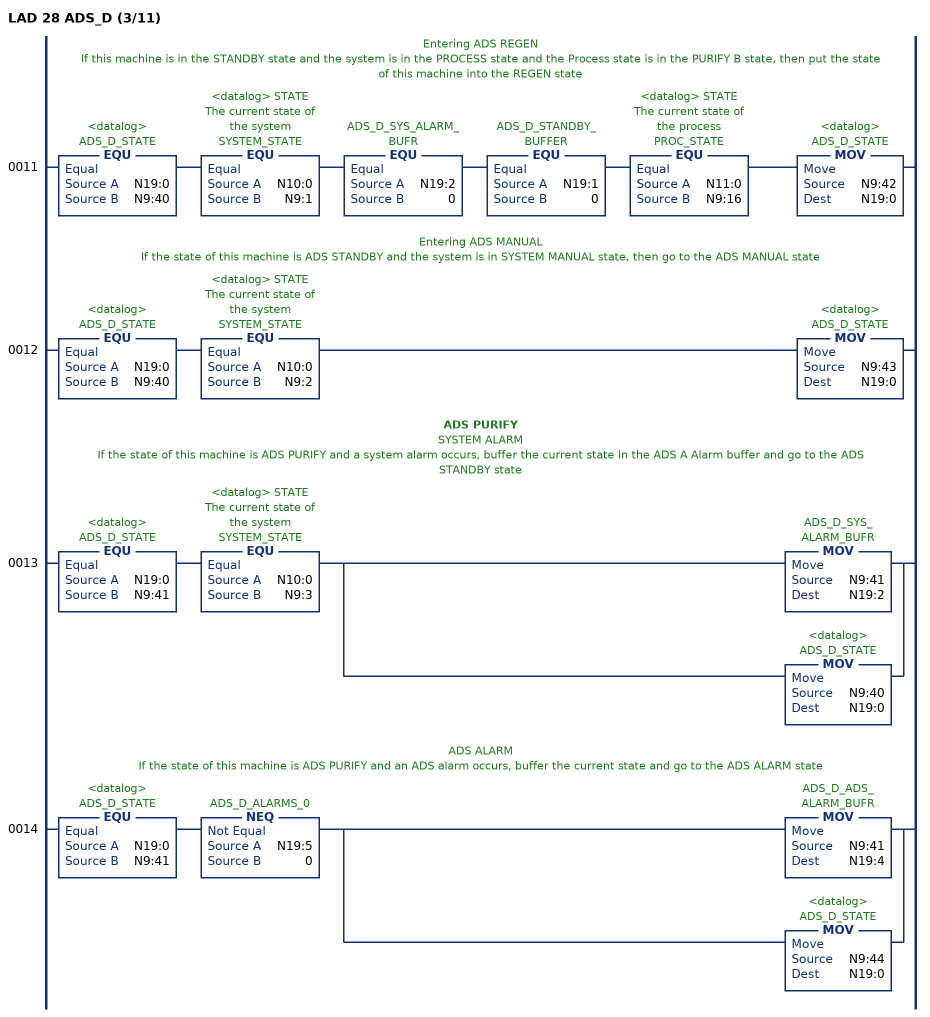
% Rung: 11 %
% Entering ADS REGEN
% If this machine is in the STANDBY state and the system is in the PROCESS state and the Process state is in the PURIFY B state, then put the state of this machine into the REGEN state %
SOR EQU N19:0 N9:40 EQU N10:0 N9:1 EQU N19:2 0 EQU N19:1 0 EQU N11:0 N9:16 MOV N9:42 N19:0 EOR
%   N19:0  ADS_D_STATE  "<datalog>" %
%   N9:40  ADS_STANDBY  "STATE ADS Standby" %
%   N10:0  SYSTEM_STATE  "<datalog> STATE The current state of the system" %
%   N9:1  SYSTEM_PROCESS  "STATE System Process" %
%   N19:2  ADS_D_SYS_ALARM_BUFR %
%   N19:1  ADS_D_STANDBY_BUFFER %
%   N11:0  PROC_STATE  "<datalog> STATE The current state of the process" %
%   N9:16  PROC_REGEN_D  "STATE Process Regen D" %
%   N9:42  ADS_REGEN  "STATE ADS Regen" %
% Rung: 12 %
% Entering ADS MANUAL
% If the state of this machine is ADS STANDBY and the system is in SYSTEM MANUAL state, then go to the ADS MANUAL state %
SOR EQU N19:0 N9:40 EQU N10:0 N9:2 MOV N9:43 N19:0 EOR
%   N19:0  ADS_D_STATE  "<datalog>" %
%   N9:40  ADS_STANDBY  "STATE ADS Standby" %
%   N10:0  SYSTEM_STATE  "<datalog> STATE The current state of the system" %
%   N9:2  SYSTEM_MANUAL  "STATE System Manual" %
%   N9:43  ADS_MANUAL  "STATE ADS Manual" %
% Rung: 13 %
% TITLE: ADS PURIFY %
% SYSTEM ALARM
% If the state of this machine is ADS PURIFY and a system alarm occurs, buffer the current state in the ADS A Alarm buffer and go to the ADS STANDBY state %
SOR EQU N19:0 N9:41 EQU N10:0 N9:3 BST MOV N9:41 N19:2 NXB MOV N9:40 N19:0 BND EOR
%   N19:0  ADS_D_STATE  "<datalog>" %
%   N9:41  ADS_PURIFY  "STATE ADS Purify" %
%   N10:0  SYSTEM_STATE  "<datalog> STATE The current state of the system" %
%   N9:3  SYSTEM_ALARM  "STATE System Alarm" %
%   N19:2  ADS_D_SYS_ALARM_BUFR %
%   N9:40  ADS_STANDBY  "STATE ADS Standby" %
% Rung: 14 %
% ADS ALARM
% If the state of this machine is ADS PURIFY and an ADS alarm occurs, buffer the current state and go to the ADS ALARM state %
SOR EQU N19:0 N9:41 NEQ N19:5 0 BST MOV N9:41 N19:4 NXB MOV N9:44 N19:0 BND EOR
%   N19:0  ADS_D_STATE  "<datalog>" %
%   N9:41  ADS_PURIFY  "STATE ADS Purify" %
%   N19:5  ADS_D_ALARMS_0 %
%   N19:4  ADS_D_ADS_ALARM_BUFR %
%   N9:44  ADS_ALARM  "STATE ADS Alarm" %

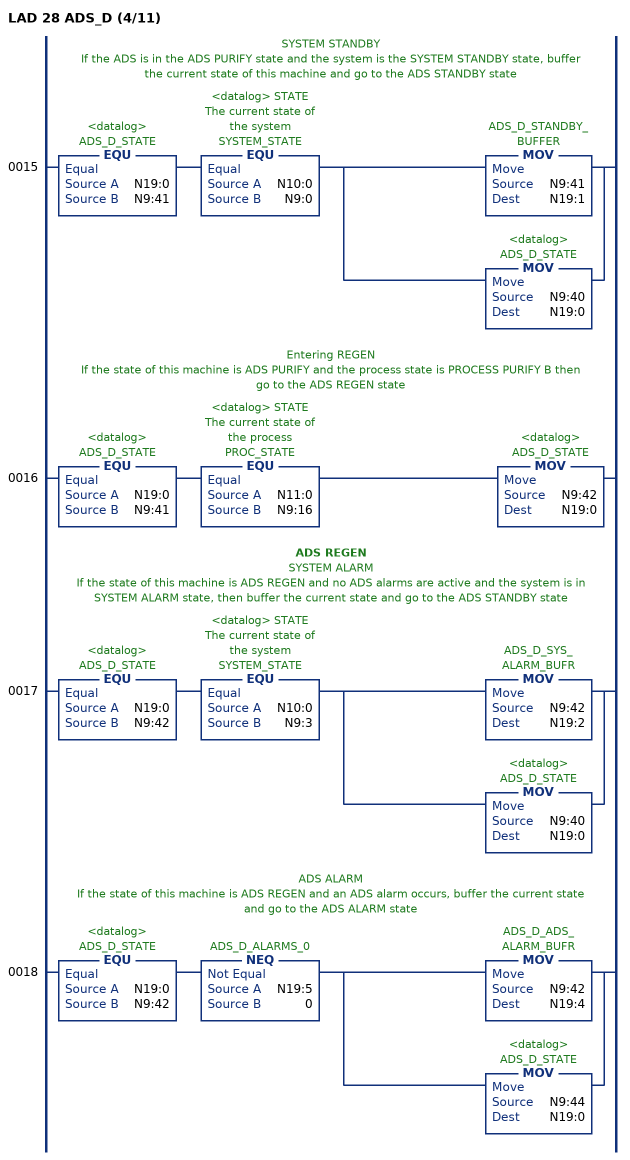
% Rung: 15 %
% SYSTEM STANDBY
% If the ADS is in the ADS PURIFY state and the system is the SYSTEM STANDBY state, buffer the current state of this machine and go to the ADS STANDBY state %
SOR EQU N19:0 N9:41 EQU N10:0 N9:0 BST MOV N9:41 N19:1 NXB MOV N9:40 N19:0 BND EOR
%   N19:0  ADS_D_STATE  "<datalog>" %
%   N9:41  ADS_PURIFY  "STATE ADS Purify" %
%   N10:0  SYSTEM_STATE  "<datalog> STATE The current state of the system" %
%   N9:0  SYSTEM_STANDBY  "STATE System Standby" %
%   N19:1  ADS_D_STANDBY_BUFFER %
%   N9:40  ADS_STANDBY  "STATE ADS Standby" %
% Rung: 16 %
% Entering REGEN
% If the state of this machine is ADS PURIFY and the process state is PROCESS PURIFY B then go to the ADS REGEN state %
SOR EQU N19:0 N9:41 EQU N11:0 N9:16 MOV N9:42 N19:0 EOR
%   N19:0  ADS_D_STATE  "<datalog>" %
%   N9:41  ADS_PURIFY  "STATE ADS Purify" %
%   N11:0  PROC_STATE  "<datalog> STATE The current state of the process" %
%   N9:16  PROC_REGEN_D  "STATE Process Regen D" %
%   N9:42  ADS_REGEN  "STATE ADS Regen" %
% Rung: 17 %
% TITLE: ADS REGEN %
% SYSTEM ALARM
% If the state of this machine is ADS REGEN and no ADS alarms are active and the system is in SYSTEM ALARM state, then buffer the current state and go to the ADS STANDBY state %
SOR EQU N19:0 N9:42 EQU N10:0 N9:3 BST MOV N9:42 N19:2 NXB MOV N9:40 N19:0 BND EOR
%   N19:0  ADS_D_STATE  "<datalog>" %
%   N9:42  ADS_REGEN  "STATE ADS Regen" %
%   N10:0  SYSTEM_STATE  "<datalog> STATE The current state of the system" %
%   N9:3  SYSTEM_ALARM  "STATE System Alarm" %
%   N19:2  ADS_D_SYS_ALARM_BUFR %
%   N9:40  ADS_STANDBY  "STATE ADS Standby" %
% Rung: 18 %
% ADS ALARM
% If the state of this machine is ADS REGEN and an ADS alarm occurs, buffer the current state and go to the ADS ALARM state %
SOR EQU N19:0 N9:42 NEQ N19:5 0 BST MOV N9:42 N19:4 NXB MOV N9:44 N19:0 BND EOR
%   N19:0  ADS_D_STATE  "<datalog>" %
%   N9:42  ADS_REGEN  "STATE ADS Regen" %
%   N19:5  ADS_D_ALARMS_0 %
%   N19:4  ADS_D_ADS_ALARM_BUFR %
%   N9:44  ADS_ALARM  "STATE ADS Alarm" %

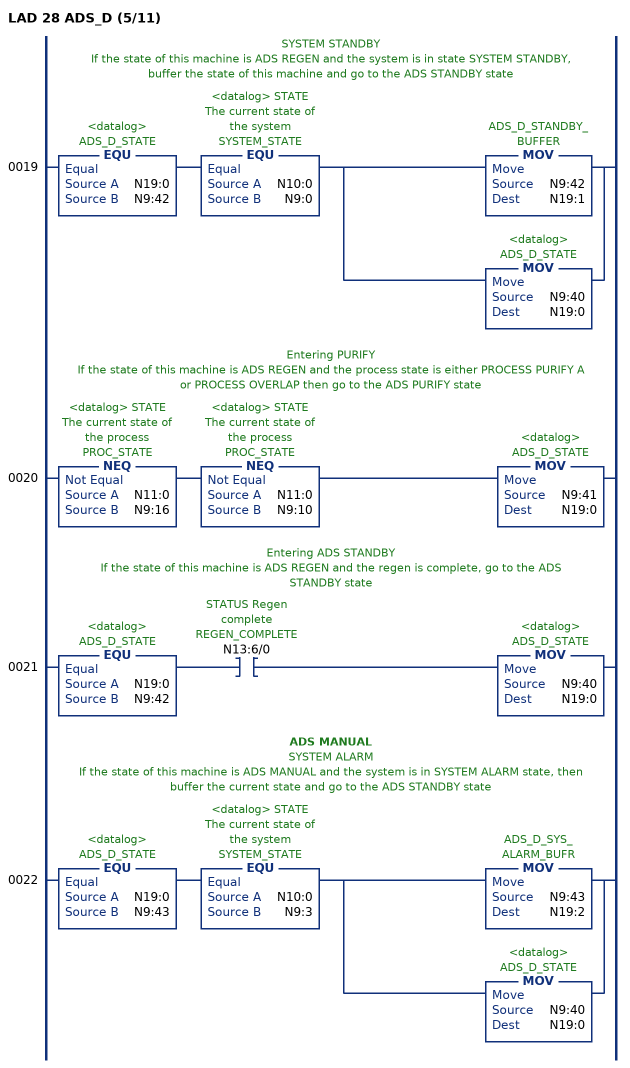
% Rung: 19 %
% SYSTEM STANDBY
% If the state of this machine is ADS REGEN and the system is in state SYSTEM STANDBY, buffer the state of this machine and go to the ADS STANDBY state %
SOR EQU N19:0 N9:42 EQU N10:0 N9:0 BST MOV N9:42 N19:1 NXB MOV N9:40 N19:0 BND EOR
%   N19:0  ADS_D_STATE  "<datalog>" %
%   N9:42  ADS_REGEN  "STATE ADS Regen" %
%   N10:0  SYSTEM_STATE  "<datalog> STATE The current state of the system" %
%   N9:0  SYSTEM_STANDBY  "STATE System Standby" %
%   N19:1  ADS_D_STANDBY_BUFFER %
%   N9:40  ADS_STANDBY  "STATE ADS Standby" %
% Rung: 20 %
% Entering PURIFY
% If the state of this machine is ADS REGEN and the process state is either PROCESS PURIFY A or PROCESS OVERLAP then go to the ADS PURIFY state %
SOR NEQ N11:0 N9:16 NEQ N11:0 N9:10 MOV N9:41 N19:0 EOR
%   N11:0  PROC_STATE  "<datalog> STATE The current state of the process" %
%   N9:16  PROC_REGEN_D  "STATE Process Regen D" %
%   N9:10  PROCESS_STANDBY  "STATE Process Standby" %
%   N9:41  ADS_PURIFY  "STATE ADS Purify" %
%   N19:0  ADS_D_STATE  "<datalog>" %
% Rung: 21 %
% Entering ADS STANDBY
% If the state of this machine is ADS REGEN and the regen is complete, go to the ADS STANDBY state %
SOR EQU N19:0 N9:42 XIC N13:6/0 MOV N9:40 N19:0 EOR
%   N19:0  ADS_D_STATE  "<datalog>" %
%   N9:42  ADS_REGEN  "STATE ADS Regen" %
%   N13:6/0  REGEN_COMPLETE  "STATUS Regen complete" %
%   N9:40  ADS_STANDBY  "STATE ADS Standby" %
% Rung: 22 %
% TITLE: ADS MANUAL %
% SYSTEM ALARM
% If the state of this machine is ADS MANUAL and the system is in SYSTEM ALARM state, then buffer the current state and go to the ADS STANDBY state %
SOR EQU N19:0 N9:43 EQU N10:0 N9:3 BST MOV N9:43 N19:2 NXB MOV N9:40 N19:0 BND EOR
%   N19:0  ADS_D_STATE  "<datalog>" %
%   N9:43  ADS_MANUAL  "STATE ADS Manual" %
%   N10:0  SYSTEM_STATE  "<datalog> STATE The current state of the system" %
%   N9:3  SYSTEM_ALARM  "STATE System Alarm" %
%   N19:2  ADS_D_SYS_ALARM_BUFR %
%   N9:40  ADS_STANDBY  "STATE ADS Standby" %

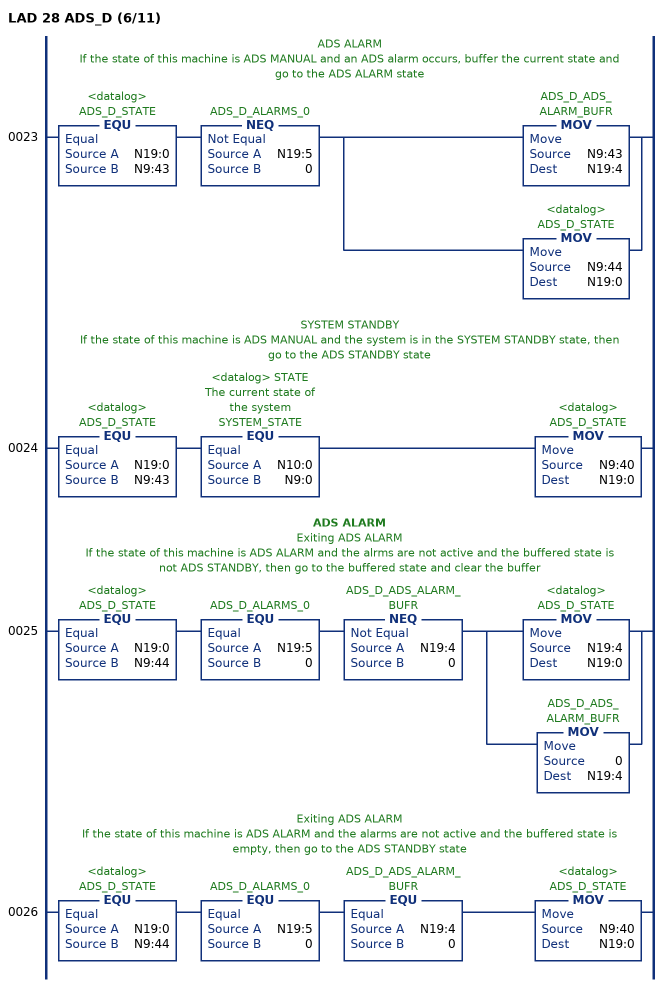
% Rung: 23 %
% ADS ALARM
% If the state of this machine is ADS MANUAL and an ADS alarm occurs, buffer the current state and go to the ADS ALARM state %
SOR EQU N19:0 N9:43 NEQ N19:5 0 BST MOV N9:43 N19:4 NXB MOV N9:44 N19:0 BND EOR
%   N19:0  ADS_D_STATE  "<datalog>" %
%   N9:43  ADS_MANUAL  "STATE ADS Manual" %
%   N19:5  ADS_D_ALARMS_0 %
%   N19:4  ADS_D_ADS_ALARM_BUFR %
%   N9:44  ADS_ALARM  "STATE ADS Alarm" %
% Rung: 24 %
% SYSTEM STANDBY
% If the state of this machine is ADS MANUAL and the system is in the SYSTEM STANDBY state, then go to the ADS STANDBY state %
SOR EQU N19:0 N9:43 EQU N10:0 N9:0 MOV N9:40 N19:0 EOR
%   N19:0  ADS_D_STATE  "<datalog>" %
%   N9:43  ADS_MANUAL  "STATE ADS Manual" %
%   N10:0  SYSTEM_STATE  "<datalog> STATE The current state of the system" %
%   N9:0  SYSTEM_STANDBY  "STATE System Standby" %
%   N9:40  ADS_STANDBY  "STATE ADS Standby" %
% Rung: 25 %
% TITLE: ADS ALARM %
% Exiting ADS ALARM
% If the state of this machine is ADS ALARM and the alrms are not active and the buffered state is not ADS STANDBY, then go to the buffered state and clear the buffer %
SOR EQU N19:0 N9:44 EQU N19:5 0 NEQ N19:4 0 BST MOV N19:4 N19:0 NXB MOV 0 N19:4 BND EOR
%   N19:0  ADS_D_STATE  "<datalog>" %
%   N9:44  ADS_ALARM  "STATE ADS Alarm" %
%   N19:5  ADS_D_ALARMS_0 %
%   N19:4  ADS_D_ADS_ALARM_BUFR %
% Rung: 26 %
% Exiting ADS ALARM
% If the state of this machine is ADS ALARM and the alarms are not active and the buffered state is empty, then go to the ADS STANDBY state %
SOR EQU N19:0 N9:44 EQU N19:5 0 EQU N19:4 0 MOV N9:40 N19:0 EOR
%   N19:0  ADS_D_STATE  "<datalog>" %
%   N9:44  ADS_ALARM  "STATE ADS Alarm" %
%   N19:5  ADS_D_ALARMS_0 %
%   N19:4  ADS_D_ADS_ALARM_BUFR %
%   N9:40  ADS_STANDBY  "STATE ADS Standby" %

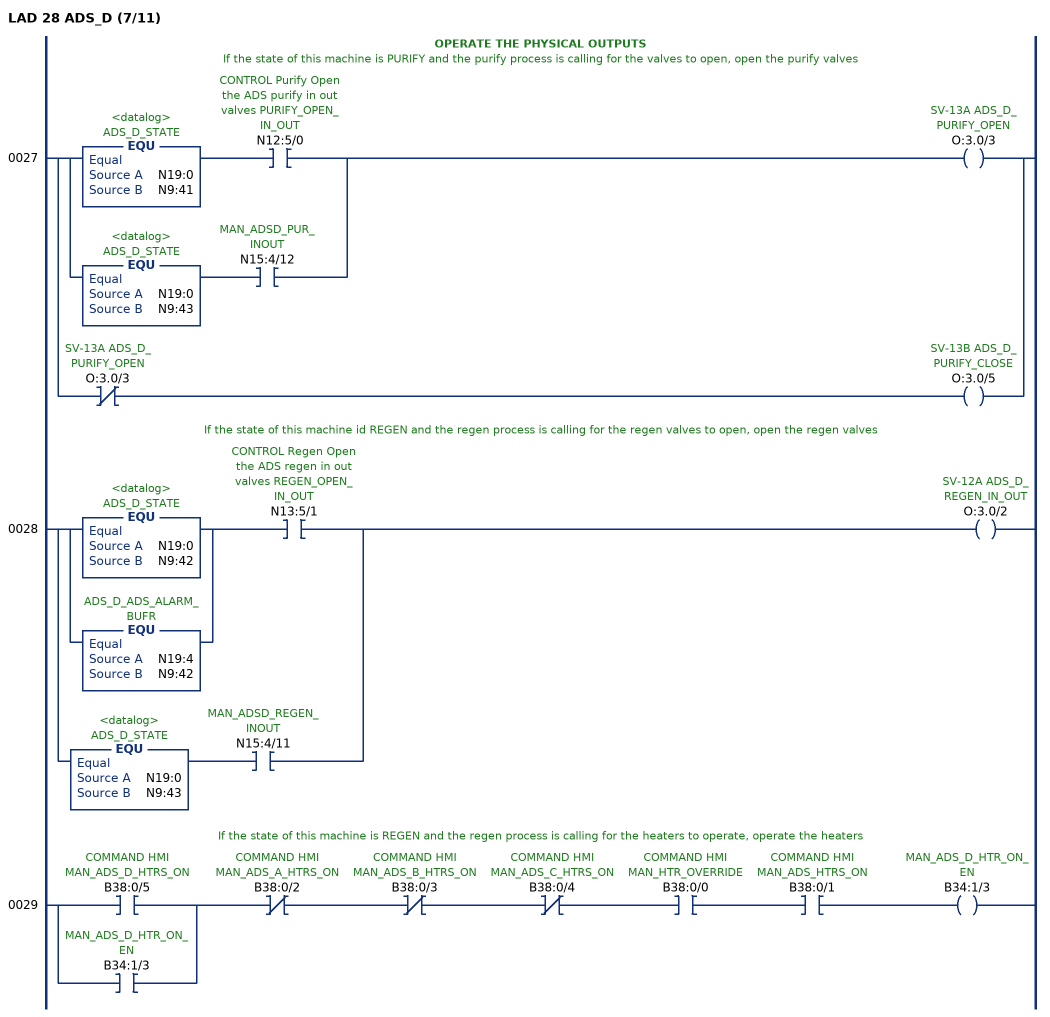
% Rung: 27 %
% TITLE: OPERATE THE PHYSICAL OUTPUTS %
% If the state of this machine is PURIFY and the purify process is calling for the valves to open, open the purify valves %
SOR BST BST EQU N19:0 N9:41 XIC N12:5/0 NXB EQU N19:0 N9:43 XIC N15:4/12 BND OTE O:3.0/3 NXB XIO O:3.0/3 OTE O:3.0/5 BND EOR
%   N19:0  ADS_D_STATE  "<datalog>" %
%   N9:41  ADS_PURIFY  "STATE ADS Purify" %
%   N12:5/0  PURIFY_OPEN_IN_OUT  "CONTROL Purify Open the ADS purify in out valves" %
%   N9:43  ADS_MANUAL  "STATE ADS Manual" %
%   N15:4/12  MAN_ADSD_PUR_INOUT %
%   O:3.0/3  ADS_D_PURIFY_OPEN  "SV-13A" %
%   O:3.0/5  ADS_D_PURIFY_CLOSE  "SV-13B" %
% Rung: 28 %
% If the state of this machine id REGEN and the regen process is calling for the regen valves to open, open the regen valves %
SOR BST BST EQU N19:0 N9:42 NXB EQU N19:4 N9:42 BND XIC N13:5/1 NXB EQU N19:0 N9:43 XIC N15:4/11 BND OTE O:3.0/2 EOR
%   N19:0  ADS_D_STATE  "<datalog>" %
%   N9:42  ADS_REGEN  "STATE ADS Regen" %
%   N19:4  ADS_D_ADS_ALARM_BUFR %
%   N13:5/1  REGEN_OPEN_IN_OUT  "CONTROL Regen Open the ADS regen in out valves" %
%   N9:43  ADS_MANUAL  "STATE ADS Manual" %
%   N15:4/11  MAN_ADSD_REGEN_INOUT %
%   O:3.0/2  ADS_D_REGEN_IN_OUT  "SV-12A" %
% Rung: 29 %
% If the state of this machine is REGEN and the regen process is calling for the heaters to operate, operate the heaters %
SOR BST XIC B38:0/5 NXB XIC B34:1/3 BND XIO B38:0/2 XIO B38:0/3 XIO B38:0/4 XIC B38:0/0 XIC B38:0/1 OTE B34:1/3 EOR
%   B38:0/5  MAN_ADS_D_HTRS_ON  "COMMAND HMI" %
%   B34:1/3  MAN_ADS_D_HTR_ON_EN %
%   B38:0/2  MAN_ADS_A_HTRS_ON  "COMMAND HMI" %
%   B38:0/3  MAN_ADS_B_HTRS_ON  "COMMAND HMI" %
%   B38:0/4  MAN_ADS_C_HTRS_ON  "COMMAND HMI" %
%   B38:0/0  MAN_HTR_OVERRIDE  "COMMAND HMI" %
%   B38:0/1  MAN_ADS_HTRS_ON  "COMMAND HMI" %

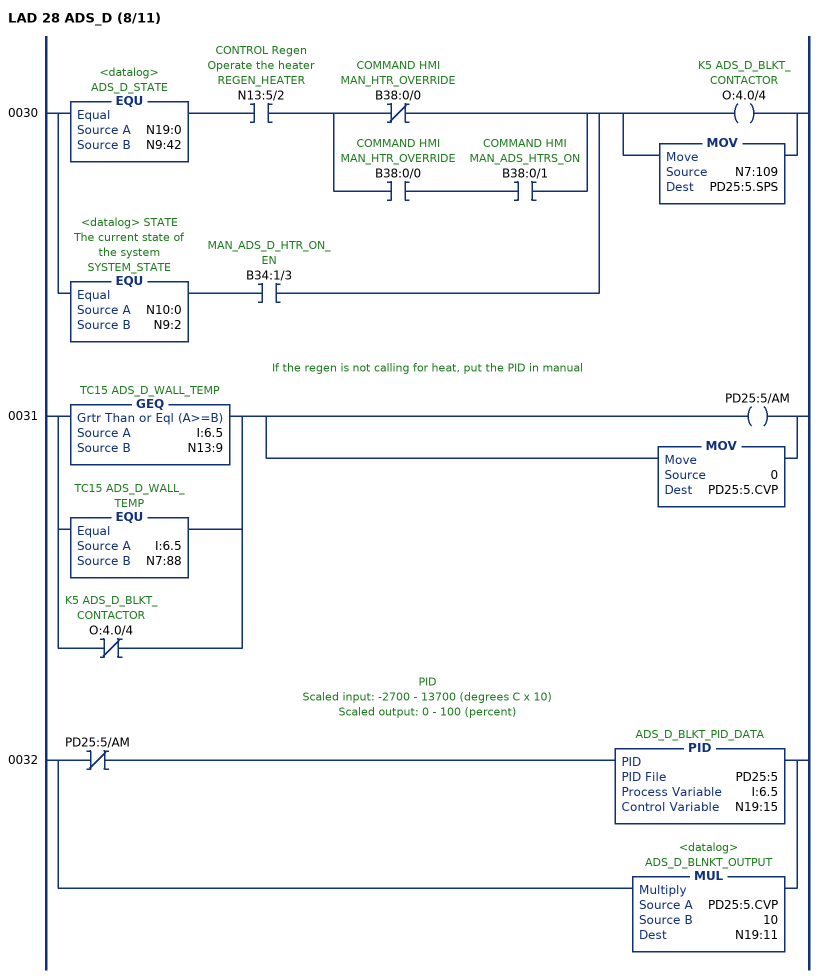
% Rung: 30 %
SOR BST EQU N19:0 N9:42 XIC N13:5/2 BST XIO B38:0/0 NXB XIC B38:0/0 XIC B38:0/1 BND NXB EQU N10:0 N9:2 XIC B34:1/3 BND BST OTE O:4.0/4 NXB MOV N7:109 PD25:5.SPS BND EOR
%   N19:0  ADS_D_STATE  "<datalog>" %
%   N9:42  ADS_REGEN  "STATE ADS Regen" %
%   N13:5/2  REGEN_HEATER  "CONTROL Regen Operate the heater" %
%   B38:0/0  MAN_HTR_OVERRIDE  "COMMAND HMI" %
%   B38:0/1  MAN_ADS_HTRS_ON  "COMMAND HMI" %
%   N10:0  SYSTEM_STATE  "<datalog> STATE The current state of the system" %
%   N9:2  SYSTEM_MANUAL  "STATE System Manual" %
%   B34:1/3  MAN_ADS_D_HTR_ON_EN %
%   O:4.0/4  ADS_D_BLKT_CONTACTOR  "K5" %
%   N7:109  BLANKET_SP  "<datalog> ADS Blanket PID Setpoint" %
% Rung: 31 %
% If the regen is not calling for heat, put the PID in manual %
SOR BST GEQ I:6.5 N13:9 NXB EQU I:6.5 N7:88 NXB XIO O:4.0/4 BND BST OTE PD25:5/AM NXB MOV 0 PD25:5.CVP BND EOR
%   I:6.5  ADS_D_WALL_TEMP  "TC15" %
%   N13:9  BLANKET_LIMIT  "ADS Blanket Temp Limit" %
%   N7:88  TC_OPEN_SP  "CONFIG TC Open Setpoint" %
%   O:4.0/4  ADS_D_BLKT_CONTACTOR  "K5" %
% Rung: 32 %
% PID
% Scaled input: -2700 - 13700 (degrees C x 10)
% Scaled output: 0 - 100 (percent) %
SOR BST XIO PD25:5/AM PID PD25:5 I:6.5 N19:15 NXB MUL PD25:5.CVP 10 N19:11 BND EOR
%   PD25:5  ADS_D_BLKT_PID_DATA %
%   I:6.5  ADS_D_WALL_TEMP  "TC15" %
%   N19:15  ADS_D_BLKT_OUTPT_RAW %
%   N19:11  ADS_D_BLNKT_OUTPUT  "<datalog>" %

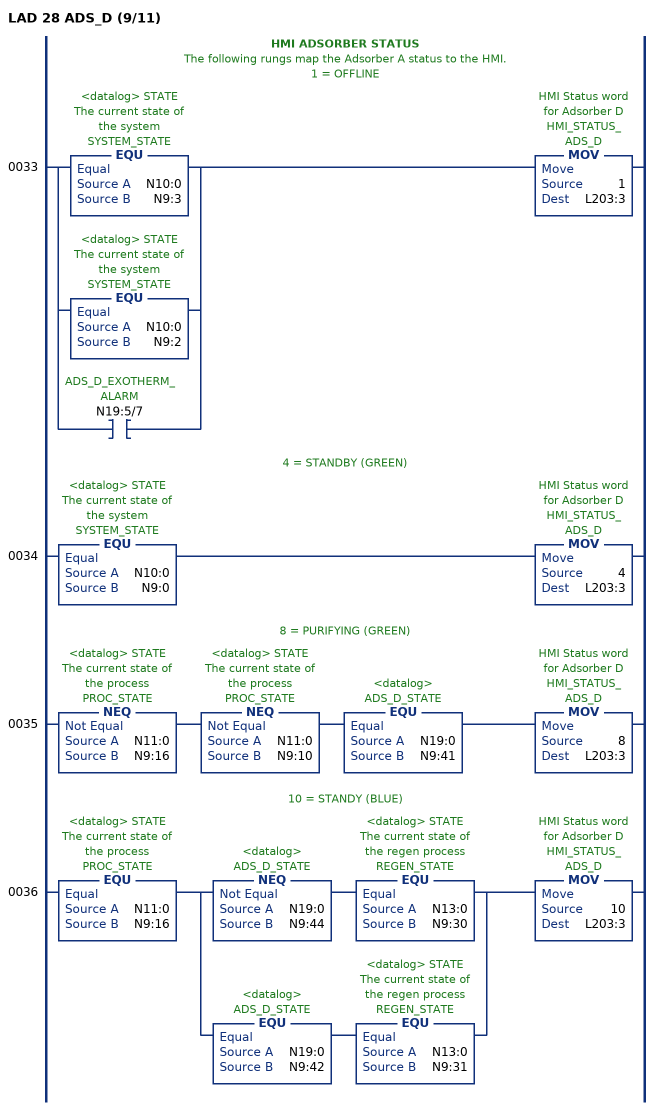
% Rung: 33 %
% TITLE: HMI ADSORBER STATUS %
% The following rungs map the Adsorber A status to the HMI.
% 1 = OFFLINE %
SOR BST EQU N10:0 N9:3 NXB EQU N10:0 N9:2 NXB XIC N19:5/7 BND MOV 1 L203:3 EOR
%   N10:0  SYSTEM_STATE  "<datalog> STATE The current state of the system" %
%   N9:3  SYSTEM_ALARM  "STATE System Alarm" %
%   N9:2  SYSTEM_MANUAL  "STATE System Manual" %
%   N19:5/7  ADS_D_EXOTHERM_ALARM %
%   L203:3  HMI_STATUS_ADS_D  "HMI Status word for Adsorber D" %
% Rung: 34 %
% 4 = STANDBY (GREEN) %
SOR EQU N10:0 N9:0 MOV 4 L203:3 EOR
%   N10:0  SYSTEM_STATE  "<datalog> STATE The current state of the system" %
%   N9:0  SYSTEM_STANDBY  "STATE System Standby" %
%   L203:3  HMI_STATUS_ADS_D  "HMI Status word for Adsorber D" %
% Rung: 35 %
% 8 = PURIFYING (GREEN) %
SOR NEQ N11:0 N9:16 NEQ N11:0 N9:10 EQU N19:0 N9:41 MOV 8 L203:3 EOR
%   N11:0  PROC_STATE  "<datalog> STATE The current state of the process" %
%   N9:16  PROC_REGEN_D  "STATE Process Regen D" %
%   N9:10  PROCESS_STANDBY  "STATE Process Standby" %
%   N19:0  ADS_D_STATE  "<datalog>" %
%   N9:41  ADS_PURIFY  "STATE ADS Purify" %
%   L203:3  HMI_STATUS_ADS_D  "HMI Status word for Adsorber D" %
% Rung: 36 %
% 10 = STANDY (BLUE) %
SOR EQU N11:0 N9:16 BST NEQ N19:0 N9:44 EQU N13:0 N9:30 NXB EQU N19:0 N9:42 EQU N13:0 N9:31 BND MOV 10 L203:3 EOR
%   N11:0  PROC_STATE  "<datalog> STATE The current state of the process" %
%   N9:16  PROC_REGEN_D  "STATE Process Regen D" %
%   N19:0  ADS_D_STATE  "<datalog>" %
%   N9:44  ADS_ALARM  "STATE ADS Alarm" %
%   N13:0  REGEN_STATE  "<datalog> STATE The current state of the regen process" %
%   N9:30  REGEN_STANDBY  "STATE Regen Standby" %
%   N9:42  ADS_REGEN  "STATE ADS Regen" %
%   N9:31  REGEN_DELAY  "STATE Regen Delay" %
%   L203:3  HMI_STATUS_ADS_D  "HMI Status word for Adsorber D" %

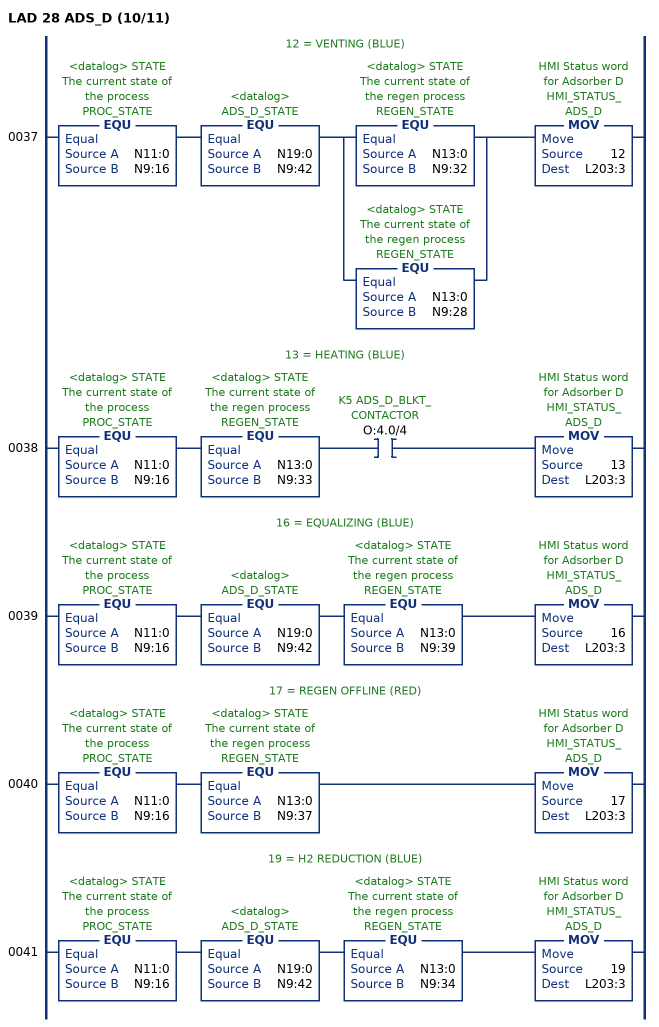
% Rung: 37 %
% 12 = VENTING (BLUE) %
SOR EQU N11:0 N9:16 EQU N19:0 N9:42 BST EQU N13:0 N9:32 NXB EQU N13:0 N9:28 BND MOV 12 L203:3 EOR
%   N11:0  PROC_STATE  "<datalog> STATE The current state of the process" %
%   N9:16  PROC_REGEN_D  "STATE Process Regen D" %
%   N19:0  ADS_D_STATE  "<datalog>" %
%   N9:42  ADS_REGEN  "STATE ADS Regen" %
%   N13:0  REGEN_STATE  "<datalog> STATE The current state of the regen process" %
%   N9:32  REGEN_VENT  "STATE Regen Vent" %
%   N9:28  REGEN_VENT_2 %
%   L203:3  HMI_STATUS_ADS_D  "HMI Status word for Adsorber D" %
% Rung: 38 %
% 13 = HEATING (BLUE) %
SOR EQU N11:0 N9:16 EQU N13:0 N9:33 XIC O:4.0/4 MOV 13 L203:3 EOR
%   N11:0  PROC_STATE  "<datalog> STATE The current state of the process" %
%   N9:16  PROC_REGEN_D  "STATE Process Regen D" %
%   N13:0  REGEN_STATE  "<datalog> STATE The current state of the regen process" %
%   N9:33  REGEN_HEAT_BED  "STATE Regen Heat wall" %
%   O:4.0/4  ADS_D_BLKT_CONTACTOR  "K5" %
%   L203:3  HMI_STATUS_ADS_D  "HMI Status word for Adsorber D" %
% Rung: 39 %
% 16 = EQUALIZING (BLUE) %
SOR EQU N11:0 N9:16 EQU N19:0 N9:42 EQU N13:0 N9:39 MOV 16 L203:3 EOR
%   N11:0  PROC_STATE  "<datalog> STATE The current state of the process" %
%   N9:16  PROC_REGEN_D  "STATE Process Regen D" %
%   N19:0  ADS_D_STATE  "<datalog>" %
%   N9:42  ADS_REGEN  "STATE ADS Regen" %
%   N13:0  REGEN_STATE  "<datalog> STATE The current state of the regen process" %
%   N9:39  REGEN_EQUALIZE  "STATE Regen Equalize" %
%   L203:3  HMI_STATUS_ADS_D  "HMI Status word for Adsorber D" %
% Rung: 40 %
% 17 = REGEN OFFLINE (RED) %
SOR EQU N11:0 N9:16 EQU N13:0 N9:37 MOV 17 L203:3 EOR
%   N11:0  PROC_STATE  "<datalog> STATE The current state of the process" %
%   N9:16  PROC_REGEN_D  "STATE Process Regen D" %
%   N13:0  REGEN_STATE  "<datalog> STATE The current state of the regen process" %
%   N9:37  REGEN_ALARM  "STATE Regen Alarm" %
%   L203:3  HMI_STATUS_ADS_D  "HMI Status word for Adsorber D" %
% Rung: 41 %
% 19 = H2 REDUCTION (BLUE) %
SOR EQU N11:0 N9:16 EQU N19:0 N9:42 EQU N13:0 N9:34 MOV 19 L203:3 EOR
%   N11:0  PROC_STATE  "<datalog> STATE The current state of the process" %
%   N9:16  PROC_REGEN_D  "STATE Process Regen D" %
%   N19:0  ADS_D_STATE  "<datalog>" %
%   N9:42  ADS_REGEN  "STATE ADS Regen" %
%   N13:0  REGEN_STATE  "<datalog> STATE The current state of the regen process" %
%   N9:34  REGEN_H2_REDUCTION  "STATE Regen Running" %
%   L203:3  HMI_STATUS_ADS_D  "HMI Status word for Adsorber D" %

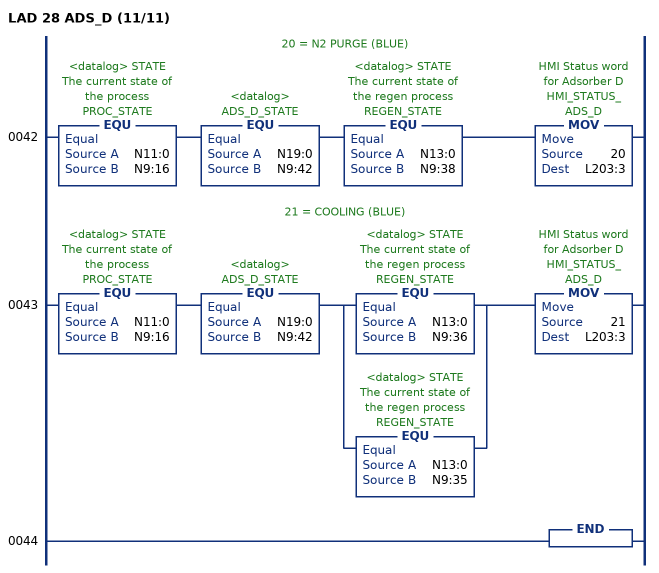
% Rung: 42 %
% 20 = N2 PURGE (BLUE) %
SOR EQU N11:0 N9:16 EQU N19:0 N9:42 EQU N13:0 N9:38 MOV 20 L203:3 EOR
%   N11:0  PROC_STATE  "<datalog> STATE The current state of the process" %
%   N9:16  PROC_REGEN_D  "STATE Process Regen D" %
%   N19:0  ADS_D_STATE  "<datalog>" %
%   N9:42  ADS_REGEN  "STATE ADS Regen" %
%   N13:0  REGEN_STATE  "<datalog> STATE The current state of the regen process" %
%   N9:38  REGEN_PURGE  "STATE Regen Hot Purge" %
%   L203:3  HMI_STATUS_ADS_D  "HMI Status word for Adsorber D" %
% Rung: 43 %
% 21 = COOLING (BLUE) %
SOR EQU N11:0 N9:16 EQU N19:0 N9:42 BST EQU N13:0 N9:36 NXB EQU N13:0 N9:35 BND MOV 21 L203:3 EOR
%   N11:0  PROC_STATE  "<datalog> STATE The current state of the process" %
%   N9:16  PROC_REGEN_D  "STATE Process Regen D" %
%   N19:0  ADS_D_STATE  "<datalog>" %
%   N9:42  ADS_REGEN  "STATE ADS Regen" %
%   N13:0  REGEN_STATE  "<datalog> STATE The current state of the regen process" %
%   N9:36  REGEN_COOL  "STATE Regen Cool" %
%   N9:35  REGEN_COOL_WALL  "STATE Regen Cool wall" %
%   L203:3  HMI_STATUS_ADS_D  "HMI Status word for Adsorber D" %
% Rung: 44 %
SOR END EOR

LADDER 29 "ADS_D_FLT"
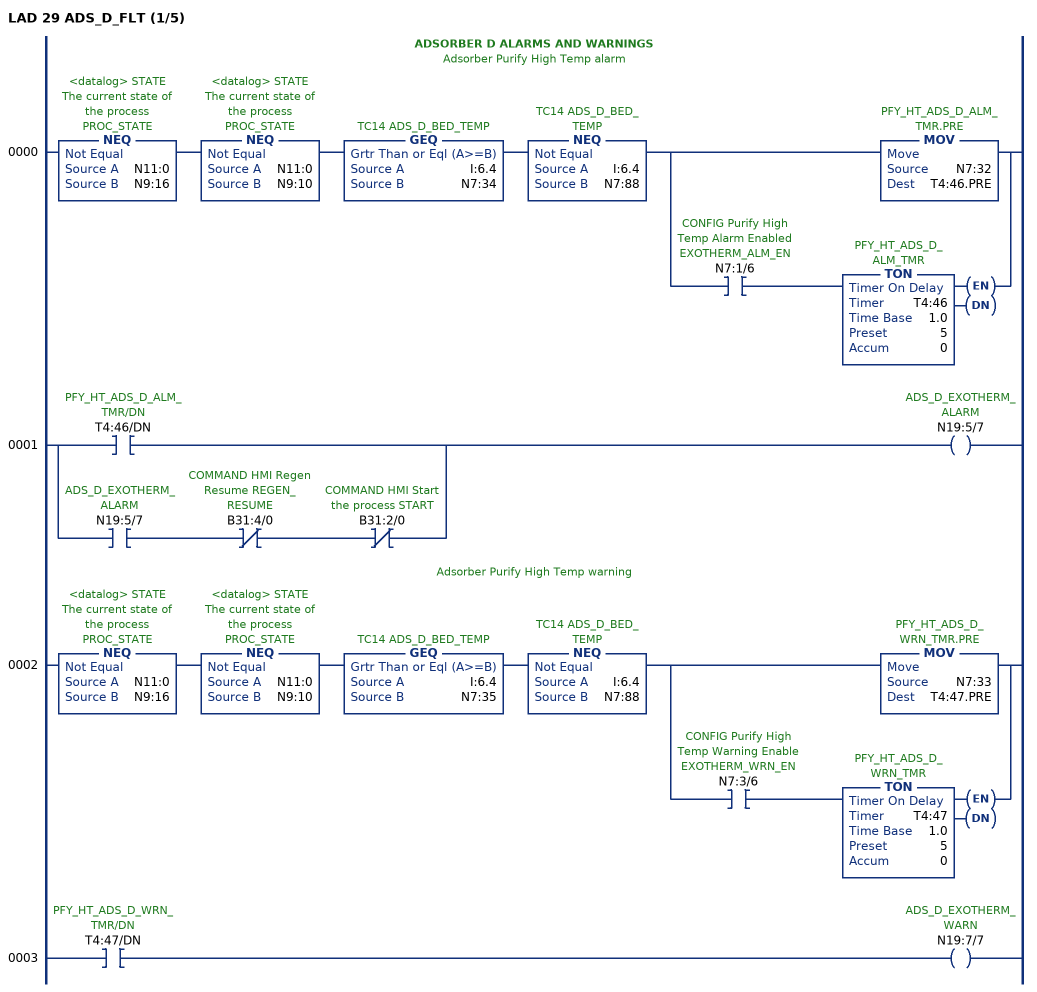
% Rung: 0 %
% TITLE: ADSORBER D ALARMS AND WARNINGS %
% Adsorber Purify High Temp alarm %
SOR NEQ N11:0 N9:16 NEQ N11:0 N9:10 GEQ I:6.4 N7:34 NEQ I:6.4 N7:88 BST MOV N7:32 T4:46.PRE NXB XIC N7:1/6 TON T4:46 1.0 5 0 BND EOR
%   N11:0  PROC_STATE  "<datalog> STATE The current state of the process" %
%   N9:16  PROC_REGEN_D  "STATE Process Regen D" %
%   N9:10  PROCESS_STANDBY  "STATE Process Standby" %
%   I:6.4  ADS_D_BED_TEMP  "TC14" %
%   N7:34  EXOTHERM_ALM_SP  "CONFIG Purify High Temp Alarm Setpoint" %
%   N7:88  TC_OPEN_SP  "CONFIG TC Open Setpoint" %
%   N7:32  EXOTHERM_ALM_DLY  "CONFIG Purify High Temp Alarm Delay" %
%   T4:46  PFY_HT_ADS_D_ALM_TMR %
%   N7:1/6  EXOTHERM_ALM_EN  "CONFIG Purify High Temp Alarm Enabled" %
% Rung: 1 %
SOR BST XIC T4:46/DN NXB XIC N19:5/7 XIO B31:4/0 XIO B31:2/0 BND OTE N19:5/7 EOR
%   T4:46  PFY_HT_ADS_D_ALM_TMR %
%   N19:5/7  ADS_D_EXOTHERM_ALARM %
%   B31:4/0  REGEN_RESUME  "COMMAND HMI Regen Resume" %
%   B31:2/0  START  "COMMAND HMI Start the process" %
% Rung: 2 %
% Adsorber Purify High Temp warning %
SOR NEQ N11:0 N9:16 NEQ N11:0 N9:10 GEQ I:6.4 N7:35 NEQ I:6.4 N7:88 BST MOV N7:33 T4:47.PRE NXB XIC N7:3/6 TON T4:47 1.0 5 0 BND EOR
%   N11:0  PROC_STATE  "<datalog> STATE The current state of the process" %
%   N9:16  PROC_REGEN_D  "STATE Process Regen D" %
%   N9:10  PROCESS_STANDBY  "STATE Process Standby" %
%   I:6.4  ADS_D_BED_TEMP  "TC14" %
%   N7:35  EXOTHERM_WRN_SP  "CONFIG Purify High Temp Warning Setpoint" %
%   N7:88  TC_OPEN_SP  "CONFIG TC Open Setpoint" %
%   N7:33  EXOTHERM_WRN_DLY  "CONFIG Purify High Temp Warning Delay" %
%   T4:47  PFY_HT_ADS_D_WRN_TMR %
%   N7:3/6  EXOTHERM_WRN_EN  "CONFIG Purify High Temp Warning Enable" %
% Rung: 3 %
SOR XIC T4:47/DN OTE N19:7/7 EOR
%   T4:47  PFY_HT_ADS_D_WRN_TMR %
%   N19:7/7  ADS_D_EXOTHERM_WARN %

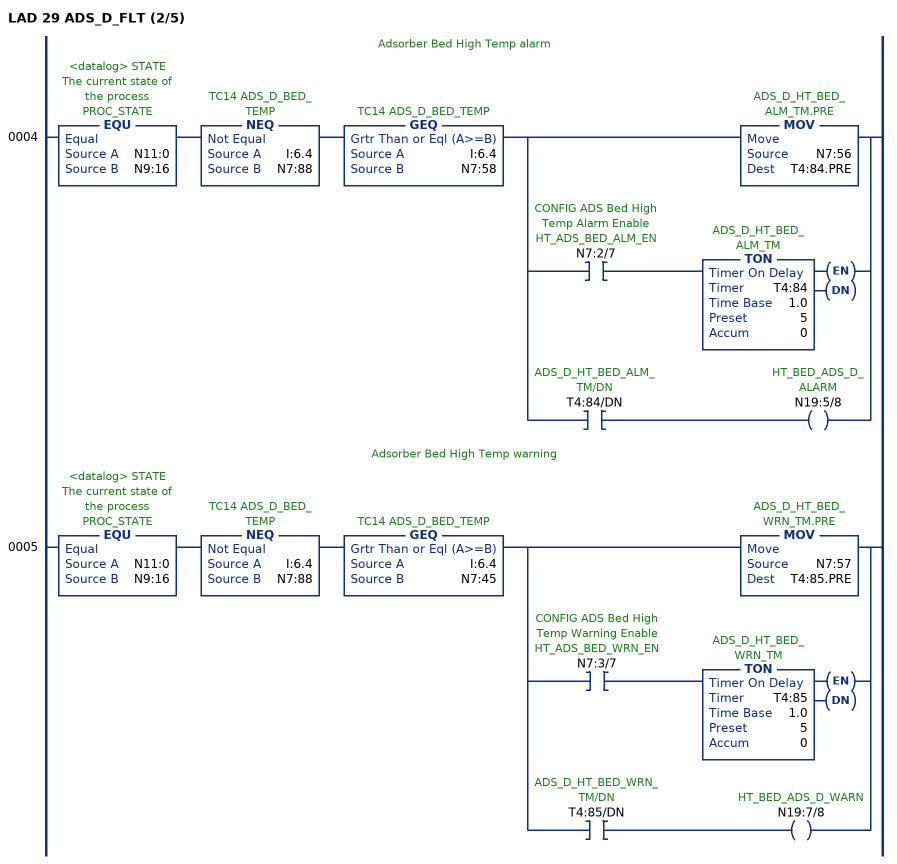
% Rung: 4 %
% Adsorber Bed High Temp alarm %
SOR EQU N11:0 N9:16 NEQ I:6.4 N7:88 GEQ I:6.4 N7:58 BST MOV N7:56 T4:84.PRE NXB XIC N7:2/7 TON T4:84 1.0 5 0 NXB XIC T4:84/DN OTE N19:5/8 BND EOR
%   N11:0  PROC_STATE  "<datalog> STATE The current state of the process" %
%   N9:16  PROC_REGEN_D  "STATE Process Regen D" %
%   I:6.4  ADS_D_BED_TEMP  "TC14" %
%   N7:88  TC_OPEN_SP  "CONFIG TC Open Setpoint" %
%   N7:58  HT_ADS_BED_ALM_SP  "CONFIG ADS Bed High Temp Alarm Setpoint" %
%   N7:56  HT_ADS_BED_ALM_DLY  "CONFIG ADS Bed High Temp Alarm Delay" %
%   T4:84  ADS_D_HT_BED_ALM_TM %
%   N7:2/7  HT_ADS_BED_ALM_EN  "CONFIG ADS Bed High Temp Alarm Enable" %
%   N19:5/8  HT_BED_ADS_D_ALARM %
% Rung: 5 %
% Adsorber Bed High Temp warning %
SOR EQU N11:0 N9:16 NEQ I:6.4 N7:88 GEQ I:6.4 N7:45 BST MOV N7:57 T4:85.PRE NXB XIC N7:3/7 TON T4:85 1.0 5 0 NXB XIC T4:85/DN OTE N19:7/8 BND EOR
%   N11:0  PROC_STATE  "<datalog> STATE The current state of the process" %
%   N9:16  PROC_REGEN_D  "STATE Process Regen D" %
%   I:6.4  ADS_D_BED_TEMP  "TC14" %
%   N7:88  TC_OPEN_SP  "CONFIG TC Open Setpoint" %
%   N7:45  LT_ADS_BED_WRN_SP  "CONFIG ADS Bed Low Temp Warning Setpoint" %
%   N7:57  HT_ADS_BED_WRN_DLY  "CONFIG ADS Bed High Temp Warning Delay" %
%   T4:85  ADS_D_HT_BED_WRN_TM %
%   N7:3/7  HT_ADS_BED_WRN_EN  "CONFIG ADS Bed High Temp Warning Enable" %
%   N19:7/8  HT_BED_ADS_D_WARN %

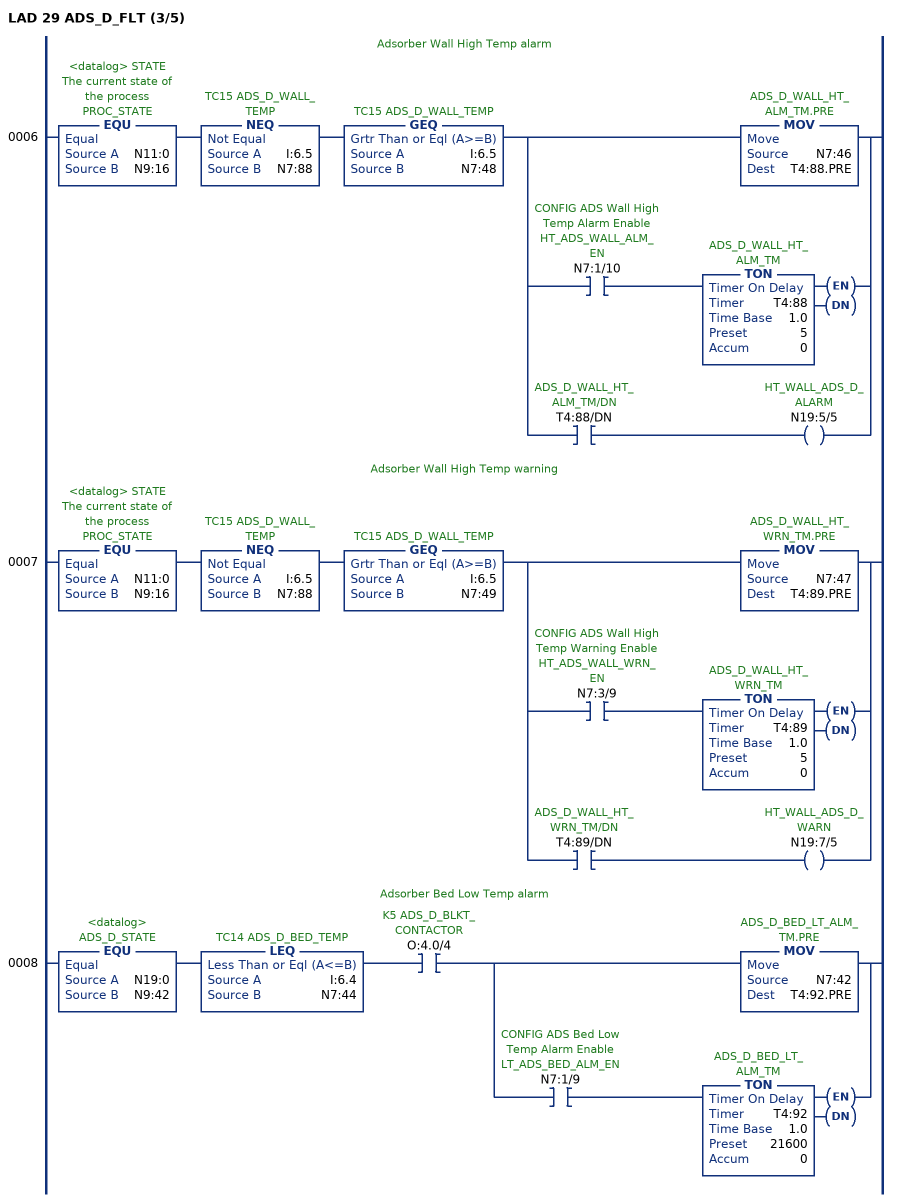
% Rung: 6 %
% Adsorber Wall High Temp alarm %
SOR EQU N11:0 N9:16 NEQ I:6.5 N7:88 GEQ I:6.5 N7:48 BST MOV N7:46 T4:88.PRE NXB XIC N7:1/10 TON T4:88 1.0 5 0 NXB XIC T4:88/DN OTE N19:5/5 BND EOR
%   N11:0  PROC_STATE  "<datalog> STATE The current state of the process" %
%   N9:16  PROC_REGEN_D  "STATE Process Regen D" %
%   I:6.5  ADS_D_WALL_TEMP  "TC15" %
%   N7:88  TC_OPEN_SP  "CONFIG TC Open Setpoint" %
%   N7:48  HT_ADS_WALL_ALM_SP  "CONFIG ADS Wall High Temp Alarm Setpoint" %
%   N7:46  HT_ADS_WALL_ALM_DLY  "CONFIG ADS Wall High Temp Alarm Delay" %
%   T4:88  ADS_D_WALL_HT_ALM_TM %
%   N7:1/10  HT_ADS_WALL_ALM_EN  "CONFIG ADS Wall High Temp Alarm Enable" %
%   N19:5/5  HT_WALL_ADS_D_ALARM %
% Rung: 7 %
% Adsorber Wall High Temp warning %
SOR EQU N11:0 N9:16 NEQ I:6.5 N7:88 GEQ I:6.5 N7:49 BST MOV N7:47 T4:89.PRE NXB XIC N7:3/9 TON T4:89 1.0 5 0 NXB XIC T4:89/DN OTE N19:7/5 BND EOR
%   N11:0  PROC_STATE  "<datalog> STATE The current state of the process" %
%   N9:16  PROC_REGEN_D  "STATE Process Regen D" %
%   I:6.5  ADS_D_WALL_TEMP  "TC15" %
%   N7:88  TC_OPEN_SP  "CONFIG TC Open Setpoint" %
%   N7:49  HT_ADS_WALL_WRN_SP  "CONFIG ADS Wall High Temp Warning Setpoint" %
%   N7:47  HT_ADS_WALL_WRN_DLY  "CONFIG ADS Wall High Temp Warning Delay" %
%   T4:89  ADS_D_WALL_HT_WRN_TM %
%   N7:3/9  HT_ADS_WALL_WRN_EN  "CONFIG ADS Wall High Temp Warning Enable" %
%   N19:7/5  HT_WALL_ADS_D_WARN %
% Rung: 8 %
% Adsorber Bed Low Temp alarm %
SOR EQU N19:0 N9:42 LEQ I:6.4 N7:44 XIC O:4.0/4 BST MOV N7:42 T4:92.PRE NXB XIC N7:1/9 TON T4:92 1.0 21600 0 BND EOR
%   N19:0  ADS_D_STATE  "<datalog>" %
%   N9:42  ADS_REGEN  "STATE ADS Regen" %
%   I:6.4  ADS_D_BED_TEMP  "TC14" %
%   N7:44  LT_ADS_BED_ALM_SP  "CONFIG ADS Bed Low Temp Alarm Setpoint" %
%   O:4.0/4  ADS_D_BLKT_CONTACTOR  "K5" %
%   N7:42  LT_ADS_BED_ALM_DLY  "CONFIG ADS Bed Low Temp Alarm Delay" %
%   T4:92  ADS_D_BED_LT_ALM_TM %
%   N7:1/9  LT_ADS_BED_ALM_EN  "CONFIG ADS Bed Low Temp Alarm Enable" %

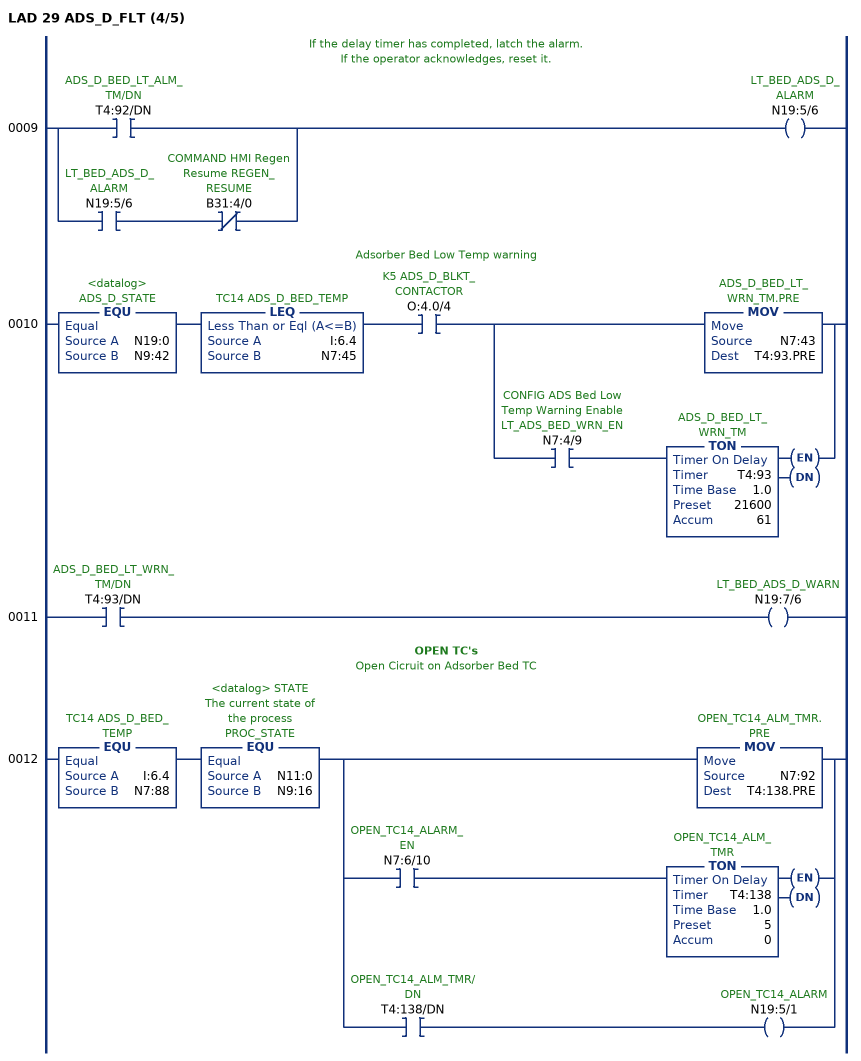
% Rung: 9 %
% If the delay timer has completed, latch the alarm.
% If the operator acknowledges, reset it. %
SOR BST XIC T4:92/DN NXB XIC N19:5/6 XIO B31:4/0 BND OTE N19:5/6 EOR
%   T4:92  ADS_D_BED_LT_ALM_TM %
%   N19:5/6  LT_BED_ADS_D_ALARM %
%   B31:4/0  REGEN_RESUME  "COMMAND HMI Regen Resume" %
% Rung: 10 %
% Adsorber Bed Low Temp warning %
SOR EQU N19:0 N9:42 LEQ I:6.4 N7:45 XIC O:4.0/4 BST MOV N7:43 T4:93.PRE NXB XIC N7:4/9 TON T4:93 1.0 21600 61 BND EOR
%   N19:0  ADS_D_STATE  "<datalog>" %
%   N9:42  ADS_REGEN  "STATE ADS Regen" %
%   I:6.4  ADS_D_BED_TEMP  "TC14" %
%   N7:45  LT_ADS_BED_WRN_SP  "CONFIG ADS Bed Low Temp Warning Setpoint" %
%   O:4.0/4  ADS_D_BLKT_CONTACTOR  "K5" %
%   N7:43  LT_ADS_BED_WRN_DLY  "CONFIG ADS Bed Low Temp Warning Delay" %
%   T4:93  ADS_D_BED_LT_WRN_TM %
%   N7:4/9  LT_ADS_BED_WRN_EN  "CONFIG ADS Bed Low Temp Warning Enable" %
% Rung: 11 %
SOR XIC T4:93/DN OTE N19:7/6 EOR
%   T4:93  ADS_D_BED_LT_WRN_TM %
%   N19:7/6  LT_BED_ADS_D_WARN %
% Rung: 12 %
% TITLE: OPEN TC's %
% Open Cicruit on Adsorber Bed TC %
SOR EQU I:6.4 N7:88 EQU N11:0 N9:16 BST MOV N7:92 T4:138.PRE NXB XIC N7:6/10 TON T4:138 1.0 5 0 NXB XIC T4:138/DN OTE N19:5/1 BND EOR
%   I:6.4  ADS_D_BED_TEMP  "TC14" %
%   N7:88  TC_OPEN_SP  "CONFIG TC Open Setpoint" %
%   N11:0  PROC_STATE  "<datalog> STATE The current state of the process" %
%   N9:16  PROC_REGEN_D  "STATE Process Regen D" %
%   N7:92  OPEN_TC_ALM_DLY  "CONFIG TC Open Alarm Delay" %
%   T4:138  OPEN_TC14_ALM_TMR %
%   N7:6/10  OPEN_TC14_ALARM_EN %
%   N19:5/1  OPEN_TC14_ALARM %

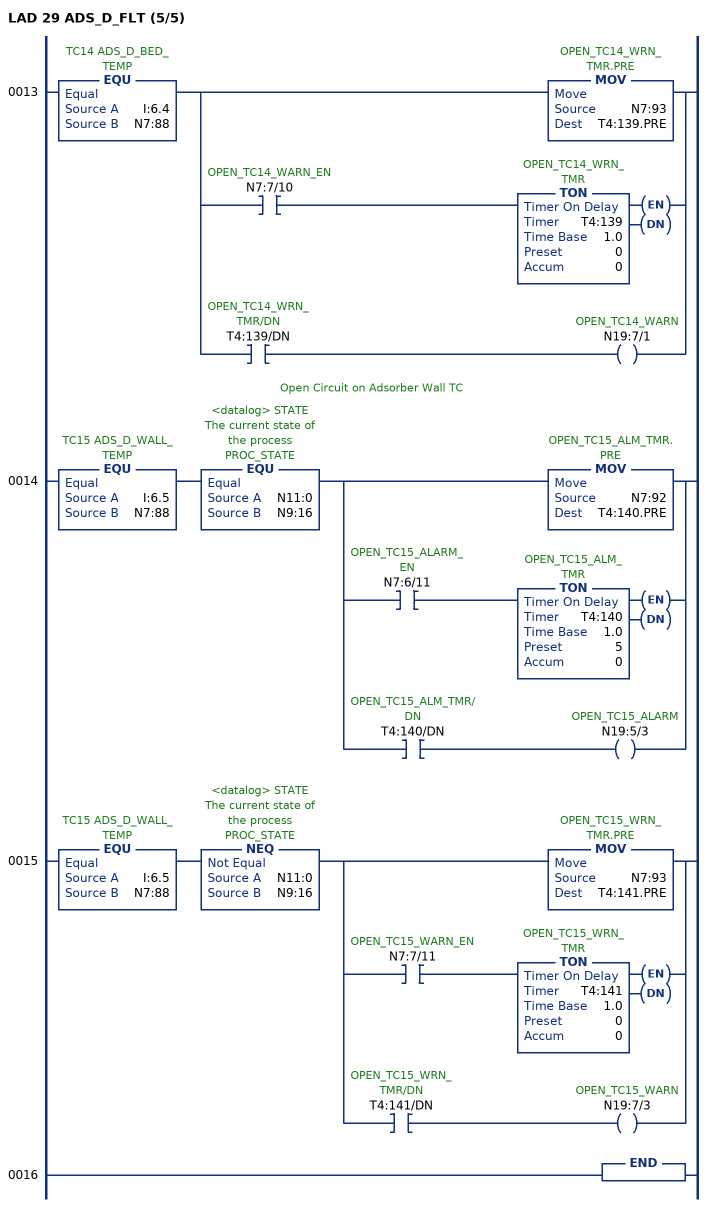
% Rung: 13 %
SOR EQU I:6.4 N7:88 BST MOV N7:93 T4:139.PRE NXB XIC N7:7/10 TON T4:139 1.0 0 0 NXB XIC T4:139/DN OTE N19:7/1 BND EOR
%   I:6.4  ADS_D_BED_TEMP  "TC14" %
%   N7:88  TC_OPEN_SP  "CONFIG TC Open Setpoint" %
%   N7:93  OPEN_TC_WRN_DLY  "CONFIG TC Open Warning Delay" %
%   T4:139  OPEN_TC14_WRN_TMR %
%   N7:7/10  OPEN_TC14_WARN_EN %
%   N19:7/1  OPEN_TC14_WARN %
% Rung: 14 %
% Open Circuit on Adsorber Wall TC %
SOR EQU I:6.5 N7:88 EQU N11:0 N9:16 BST MOV N7:92 T4:140.PRE NXB XIC N7:6/11 TON T4:140 1.0 5 0 NXB XIC T4:140/DN OTE N19:5/3 BND EOR
%   I:6.5  ADS_D_WALL_TEMP  "TC15" %
%   N7:88  TC_OPEN_SP  "CONFIG TC Open Setpoint" %
%   N11:0  PROC_STATE  "<datalog> STATE The current state of the process" %
%   N9:16  PROC_REGEN_D  "STATE Process Regen D" %
%   N7:92  OPEN_TC_ALM_DLY  "CONFIG TC Open Alarm Delay" %
%   T4:140  OPEN_TC15_ALM_TMR %
%   N7:6/11  OPEN_TC15_ALARM_EN %
%   N19:5/3  OPEN_TC15_ALARM %
% Rung: 15 %
SOR EQU I:6.5 N7:88 NEQ N11:0 N9:16 BST MOV N7:93 T4:141.PRE NXB XIC N7:7/11 TON T4:141 1.0 0 0 NXB XIC T4:141/DN OTE N19:7/3 BND EOR
%   I:6.5  ADS_D_WALL_TEMP  "TC15" %
%   N7:88  TC_OPEN_SP  "CONFIG TC Open Setpoint" %
%   N11:0  PROC_STATE  "<datalog> STATE The current state of the process" %
%   N9:16  PROC_REGEN_D  "STATE Process Regen D" %
%   N7:93  OPEN_TC_WRN_DLY  "CONFIG TC Open Warning Delay" %
%   T4:141  OPEN_TC15_WRN_TMR %
%   N7:7/11  OPEN_TC15_WARN_EN %
%   N19:7/3  OPEN_TC15_WARN %
% Rung: 16 %
SOR END EOR

LADDER 49 "MODBUS"
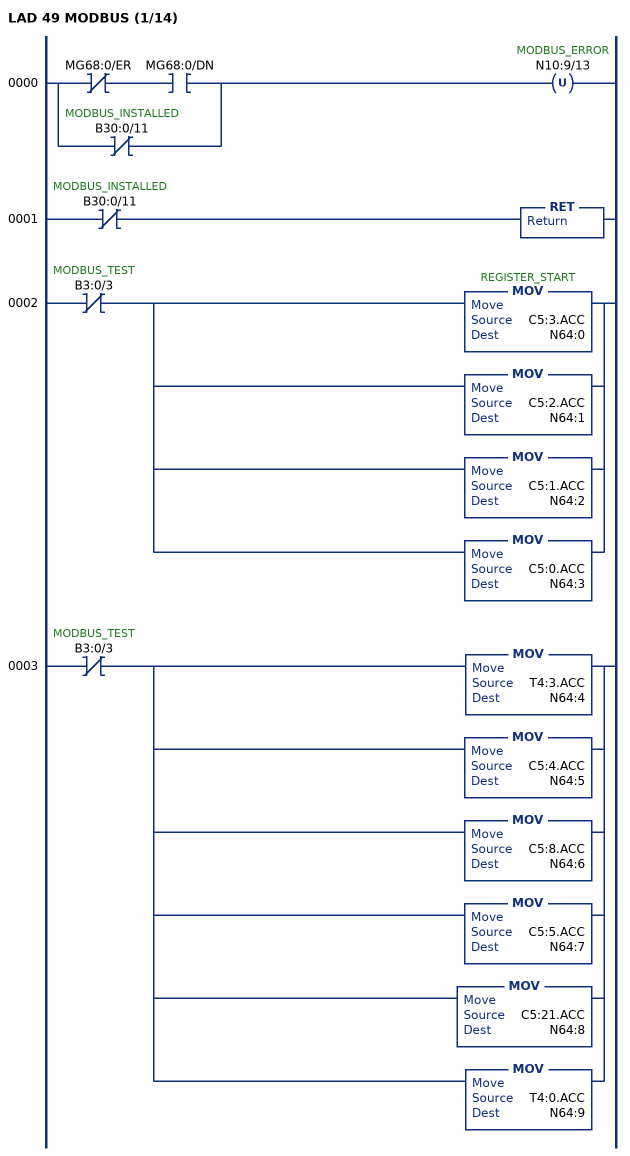
% Rung: 0 %
SOR BST XIO MG68:0/ER XIC MG68:0/DN NXB XIO B30:0/11 BND OTU N10:9/13 EOR
%   B30:0/11  MODBUS_INSTALLED %
%   N10:9/13  MODBUS_ERROR %
% Rung: 1 %
SOR XIO B30:0/11 RET EOR
%   B30:0/11  MODBUS_INSTALLED %
% Rung: 2 %
SOR XIO B3:0/3 BST MOV C5:3.ACC N64:0 NXB MOV C5:2.ACC N64:1 NXB MOV C5:1.ACC N64:2 NXB MOV C5:0.ACC N64:3 BND EOR
%   B3:0/3  MODBUS_TEST %
%   C5:3  PURIFY_ACTIVE_TTL_DY  "COUNTER The number of total elapsed purification days for the process equipment" %
%   N64:0  REGISTER_START %
%   C5:2  PURIFY_ACTIVE_TTL_HR  "COUNTER The number of total elapsed purification hours for the process equipment" %
%   C5:1  PURIFY_ACTIVE_MINUTE  "COUNTER The number of elapsed purification minutes for the current ADS (60 min)" %
%   C5:0  PURIFY_ACTIVE_HOURS  "COUNTER The number of elapsed purification hours for the current ADS" %
% Rung: 3 %
SOR XIO B3:0/3 BST MOV T4:3.ACC N64:4 NXB MOV C5:4.ACC N64:5 NXB MOV C5:8.ACC N64:6 NXB MOV C5:5.ACC N64:7 NXB MOV C5:21.ACC N64:8 NXB MOV T4:0.ACC N64:9 BND EOR
%   B3:0/3  MODBUS_TEST %
%   T4:3  REGEN_VENT_TIMER  "TIMER Regen Vent (seconds)" %
%   C5:4  REGEN_REDUC_MINUTE  "COUNTER Regen The number of minutes which the regen reduc runs" %
%   C5:8  REGEN_PURGE_MINUTES  "COUNTER Regen THe number of minutes the purge step runs" %
%   C5:5  REGEN_COOL_MINUTE  "COUNTER Regen the number of minutes for which the bed has cooled" %
%   C5:21  REGEN_EQUALIZE_MIN %
%   T4:0  PURIFY_OVERLAP_TIMER  "TIMER Purify Overlap" %

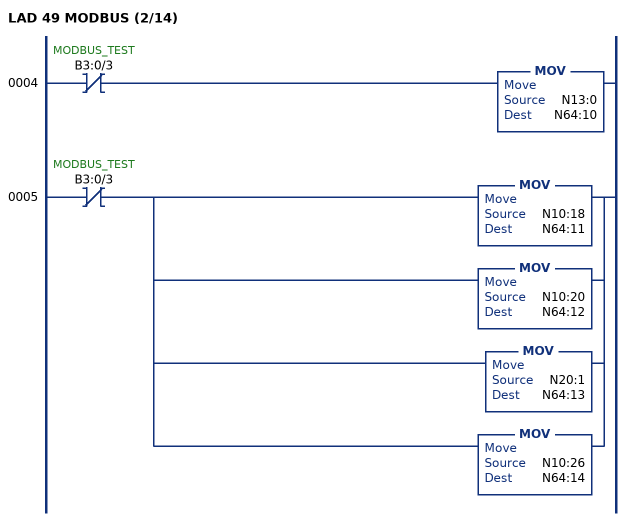
% Rung: 4 %
SOR XIO B3:0/3 MOV N13:0 N64:10 EOR
%   B3:0/3  MODBUS_TEST %
%   N13:0  REGEN_STATE  "<datalog> STATE The current state of the regen process" %
% Rung: 5 %
SOR XIO B3:0/3 BST MOV N10:18 N64:11 NXB MOV N10:20 N64:12 NXB MOV N20:1 N64:13 NXB MOV N10:26 N64:14 BND EOR
%   B3:0/3  MODBUS_TEST %
%   N10:18  INLET_PX_PSIG %
%   N10:20  OUTLET_PX_PSIG %
%   N20:1  MIX_PANEL_PSIG  "<datalog>" %
%   N10:26  MFM_FLOW  "<datalog>" %

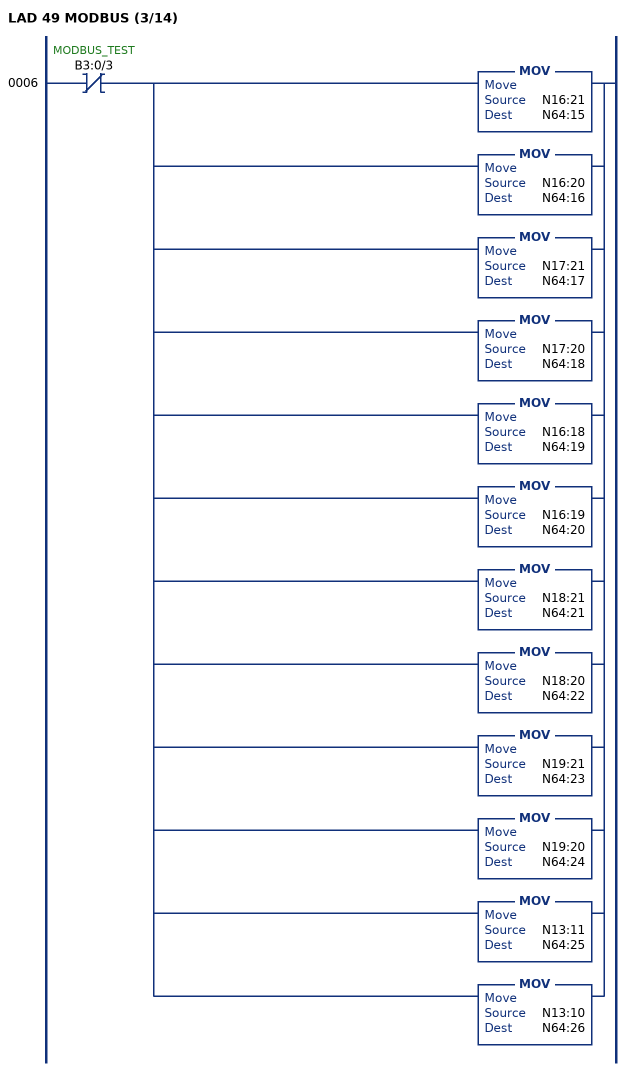
% Rung: 6 %
SOR XIO B3:0/3 BST MOV N16:21 N64:15 NXB MOV N16:20 N64:16 NXB MOV N17:21 N64:17 NXB MOV N17:20 N64:18 NXB MOV N16:18 N64:19 NXB MOV N16:19 N64:20 NXB MOV N18:21 N64:21 NXB MOV N18:20 N64:22 NXB MOV N19:21 N64:23 NXB MOV N19:20 N64:24 NXB MOV N13:11 N64:25 NXB MOV N13:10 N64:26 BND EOR
%   B3:0/3  MODBUS_TEST %
%   N16:21  ADS_A_BED_TEMP_READ  "<datalog>" %
%   N16:20  ADS_A_WALL_TEMP_READ  "<datalog>" %
%   N17:21  ADS_B_BED_TEMP_READ  "<datalog>" %
%   N17:20  ADS_B_WALL_TEMP_READ  "<datalog>" %
%   N16:18  ADS_PH_GAS_TEMP_READ  "<datalog>" %
%   N16:19  ADS_PH_ROD_TEMP_READ  "<datalog>" %
%   N18:21  ADS_C_BED_TEMP_READ  "<datalog>" %
%   N18:20  ADS_C_WALL_TEMP_READ  "<datalog>" %
%   N19:21  ADS_D_BED_TEMP_READ  "<datalog>" %
%   N19:20  ADS_D_WALL_TEMP_READ  "<datalog>" %
%   N13:11  REGEN_HRS_LEFT %
%   N13:10  REGEN_MIN_LEFT %

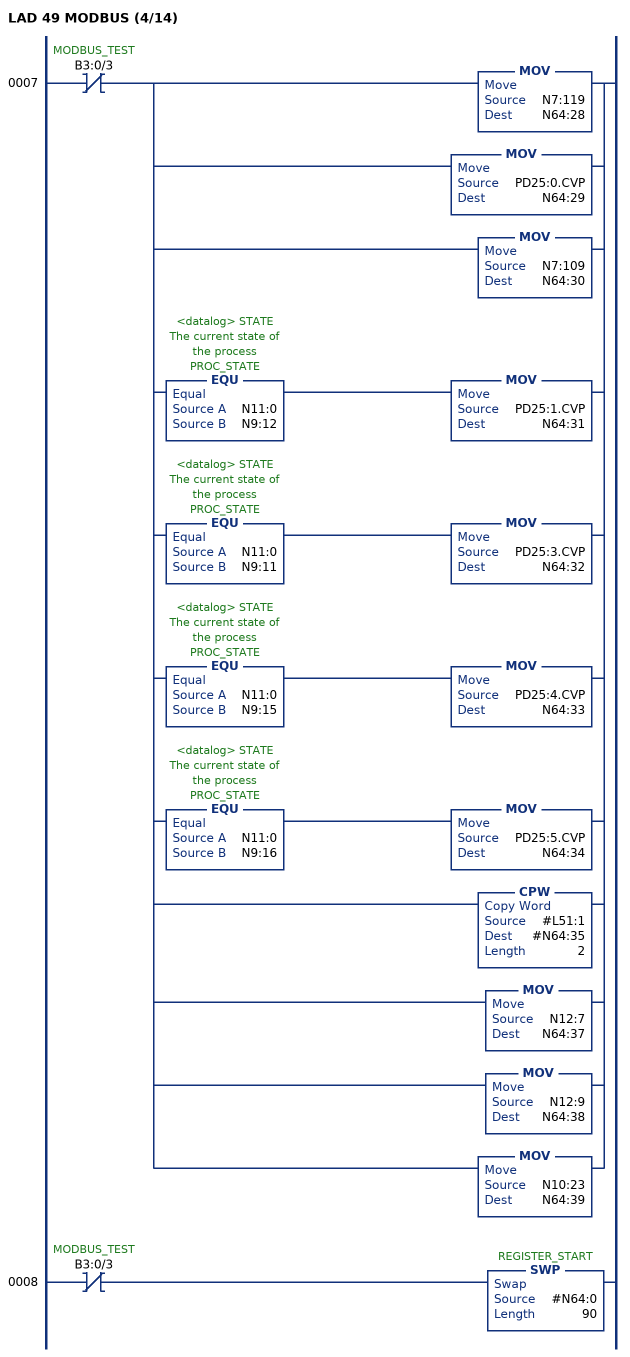
% Rung: 7 %
SOR XIO B3:0/3 BST MOV N7:119 N64:28 NXB MOV PD25:0.CVP N64:29 NXB MOV N7:109 N64:30 NXB EQU N11:0 N9:12 MOV PD25:1.CVP N64:31 NXB EQU N11:0 N9:11 MOV PD25:3.CVP N64:32 NXB EQU N11:0 N9:15 MOV PD25:4.CVP N64:33 NXB EQU N11:0 N9:16 MOV PD25:5.CVP N64:34 NXB CPW #L51:1 #N64:35 2 NXB MOV N12:7 N64:37 NXB MOV N12:9 N64:38 NXB MOV N10:23 N64:39 BND EOR
%   B3:0/3  MODBUS_TEST %
%   N7:119  PREHEATER_SP  "<datalog> ADS Preheater PID Setpoint" %
%   N7:109  BLANKET_SP  "<datalog> ADS Blanket PID Setpoint" %
%   N11:0  PROC_STATE  "<datalog> STATE The current state of the process" %
%   N9:12  PROC_REGEN_A  "STATE Process Regen A" %
%   N9:11  PROC_REGEN_B  "STATE Process Regen B" %
%   N9:15  PROC_REGEN_C  "STATE Process Regen C" %
%   N9:16  PROC_REGEN_D  "STATE Process Regen D" %
%   L51:1  TOTAL_FLOW %
%   N12:7  HOURS_LEFT_IN_PURIFY %
%   N12:9  MIN_LEFT_IN_PURIFY %
%   N10:23  H2_SENSOR_LEVEL %
% Rung: 8 %
SOR XIO B3:0/3 SWP #N64:0 90 EOR
%   B3:0/3  MODBUS_TEST %
%   N64:0  REGISTER_START %

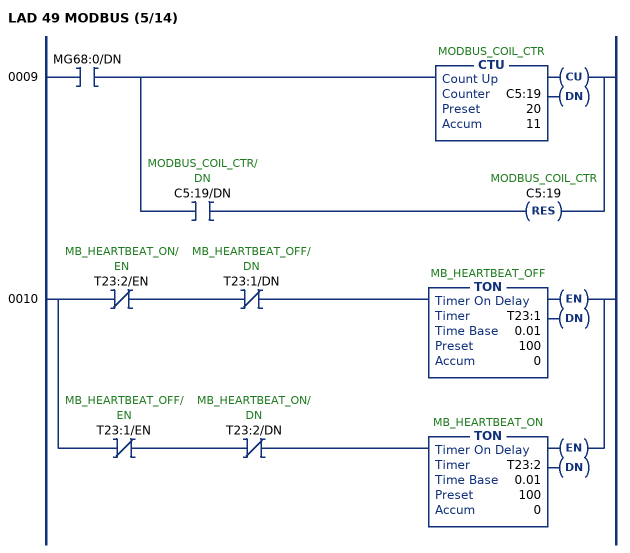
% Rung: 9 %
SOR XIC MG68:0/DN BST CTU C5:19 20 11 NXB XIC C5:19/DN RES C5:19 BND EOR
%   C5:19  MODBUS_COIL_CTR %
% Rung: 10 %
SOR BST XIO T23:2/EN XIO T23:1/DN TON T23:1 0.01 100 0 NXB XIO T23:1/EN XIO T23:2/DN TON T23:2 0.01 100 0 BND EOR
%   T23:2  MB_HEARTBEAT_ON %
%   T23:1  MB_HEARTBEAT_OFF %

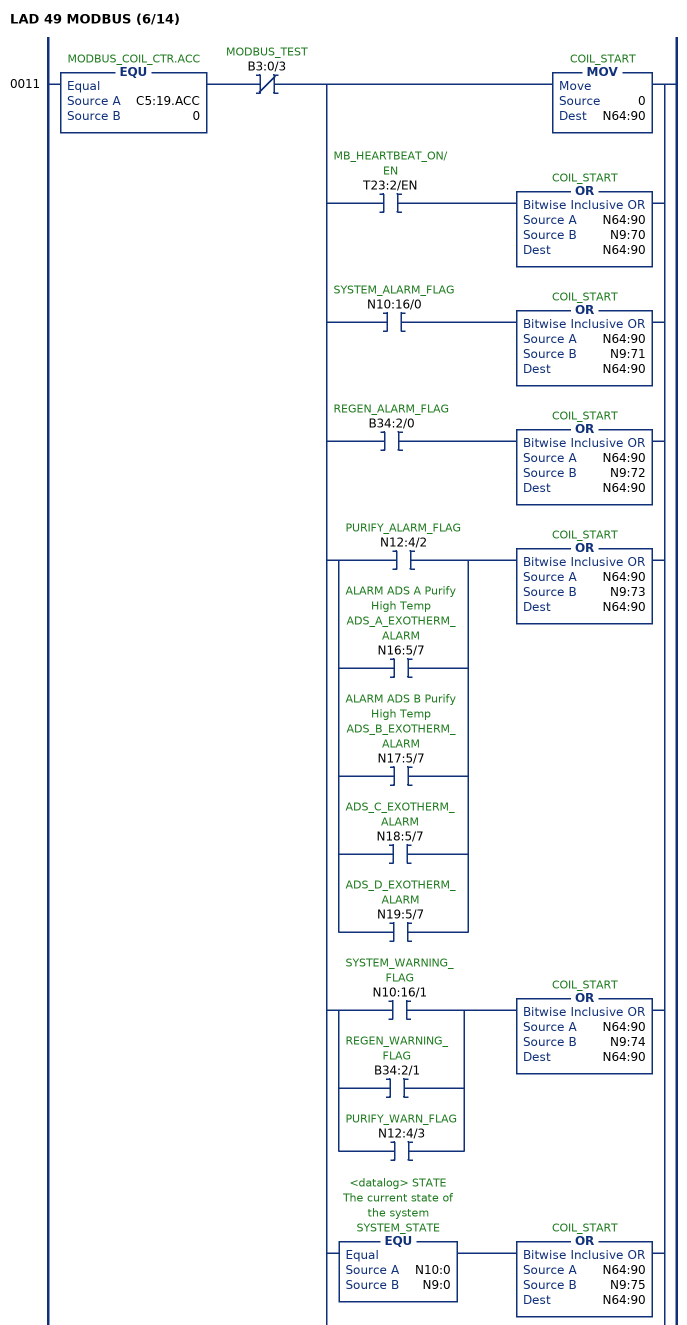

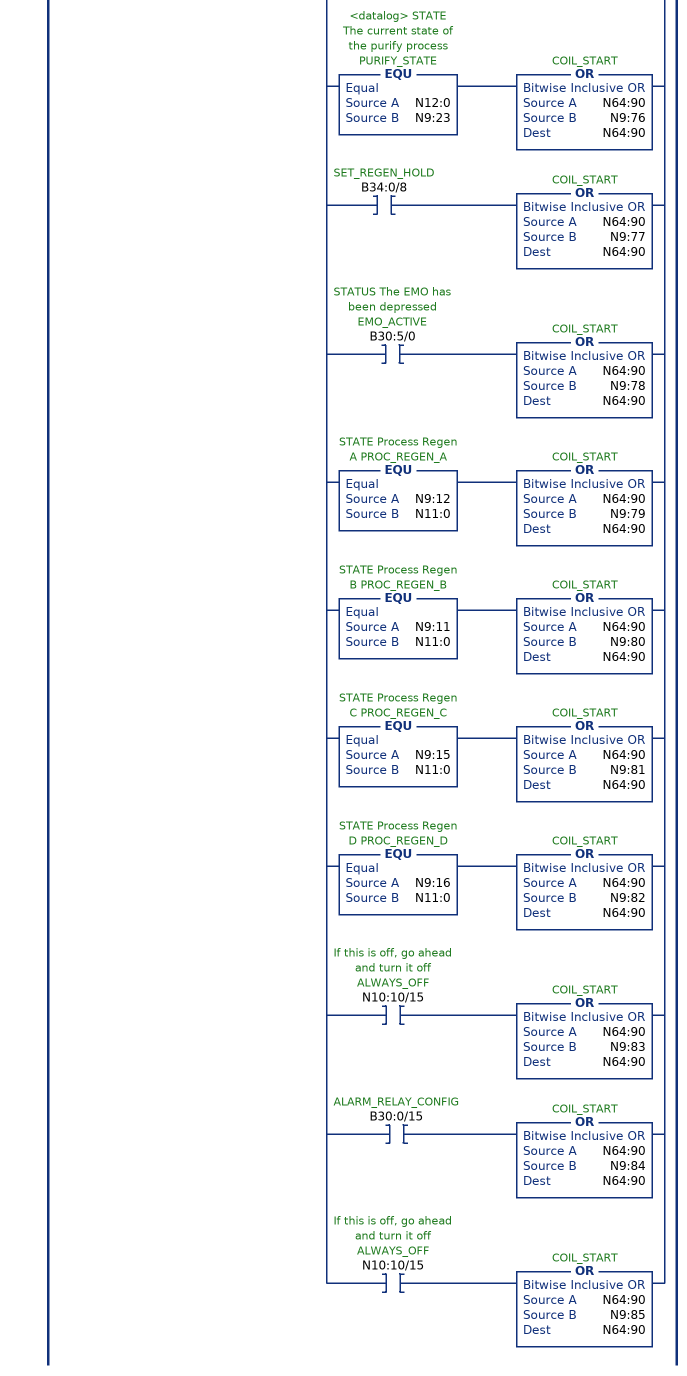
% Rung: 11 %
SOR EQU C5:19.ACC 0 XIO B3:0/3 BST MOV 0 N64:90 NXB XIC T23:2/EN OR N64:90 N9:70 N64:90 NXB XIC N10:16/0 OR N64:90 N9:71 N64:90 NXB XIC B34:2/0 OR N64:90 N9:72 N64:90 NXB BST XIC N12:4/2 NXB XIC N16:5/7 NXB XIC N17:5/7 NXB XIC N18:5/7 NXB XIC N19:5/7 BND OR N64:90 N9:73 N64:90 NXB BST XIC N10:16/1 NXB XIC B34:2/1 NXB XIC N12:4/3 BND OR N64:90 N9:74 N64:90 NXB EQU N10:0 N9:0 OR N64:90 N9:75 N64:90 NXB EQU N12:0 N9:23 OR N64:90 N9:76 N64:90 NXB XIC B34:0/8 OR N64:90 N9:77 N64:90 NXB XIC B30:5/0 OR N64:90 N9:78 N64:90 NXB EQU N9:12 N11:0 OR N64:90 N9:79 N64:90 NXB EQU N9:11 N11:0 OR N64:90 N9:80 N64:90 NXB EQU N9:15 N11:0 OR N64:90 N9:81 N64:90 NXB EQU N9:16 N11:0 OR N64:90 N9:82 N64:90 NXB XIC N10:10/15 OR N64:90 N9:83 N64:90 NXB XIC B30:0/15 OR N64:90 N9:84 N64:90 NXB XIC N10:10/15 OR N64:90 N9:85 N64:90 BND EOR
%   C5:19  MODBUS_COIL_CTR %
%   B3:0/3  MODBUS_TEST %
%   N64:90  COIL_START %
%   T23:2  MB_HEARTBEAT_ON %
%   N9:70  BIT_0 %
%   N10:16/0  SYSTEM_ALARM_FLAG %
%   N9:71  BIT_1 %
%   B34:2/0  REGEN_ALARM_FLAG %
%   N9:72  BIT_2 %
%   N12:4/2  PURIFY_ALARM_FLAG %
%   N16:5/7  ADS_A_EXOTHERM_ALARM  "ALARM ADS A Purify High Temp" %
%   N17:5/7  ADS_B_EXOTHERM_ALARM  "ALARM ADS B Purify High Temp" %
%   N18:5/7  ADS_C_EXOTHERM_ALARM %
%   N19:5/7  ADS_D_EXOTHERM_ALARM %
%   N9:73  BIT_3 %
%   N10:16/1  SYSTEM_WARNING_FLAG %
%   B34:2/1  REGEN_WARNING_FLAG %
%   N12:4/3  PURIFY_WARN_FLAG %
%   N9:74  BIT_4 %
%   N10:0  SYSTEM_STATE  "<datalog> STATE The current state of the system" %
%   N9:0  SYSTEM_STANDBY  "STATE System Standby" %
%   N9:75  BIT_5 %
%   N12:0  PURIFY_STATE  "<datalog> STATE The current state of the purify process" %
%   N9:23  PURIFY_MANUAL_HOLD  "STATE Purify Manual Hold" %
%   N9:76  BIT_6 %
%   B34:0/8  SET_REGEN_HOLD %
%   N9:77  BIT_7 %
%   B30:5/0  EMO_ACTIVE  "STATUS The EMO has been depressed" %
%   N9:78  BIT_8 %
%   N9:12  PROC_REGEN_A  "STATE Process Regen A" %
%   N11:0  PROC_STATE  "<datalog> STATE The current state of the process" %
%   N9:79  BIT_9 %
%   N9:11  PROC_REGEN_B  "STATE Process Regen B" %
%   N9:80  BIT_10 %
%   N9:15  PROC_REGEN_C  "STATE Process Regen C" %
%   N9:81  BIT_11 %
%   N9:16  PROC_REGEN_D  "STATE Process Regen D" %
%   N9:82  BIT_12 %
%   N10:10/15  ALWAYS_OFF  "If this is off, go ahead and turn it off" %
%   N9:83  BIT_13 %
%   B30:0/15  ALARM_RELAY_CONFIG %
%   N9:84  BIT_14 %
%   N9:85  BIT_15 %

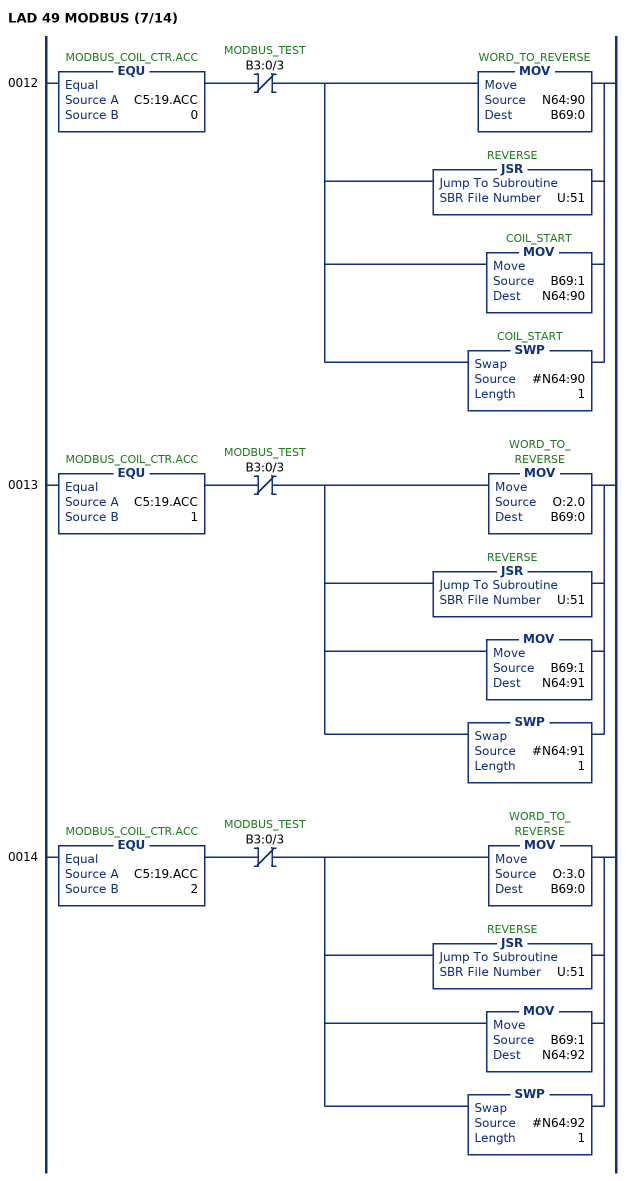
% Rung: 12 %
SOR EQU C5:19.ACC 0 XIO B3:0/3 BST MOV N64:90 B69:0 NXB JSR U:51 NXB MOV B69:1 N64:90 NXB SWP #N64:90 1 BND EOR
%   C5:19  MODBUS_COIL_CTR %
%   B3:0/3  MODBUS_TEST %
%   N64:90  COIL_START %
%   B69:0  WORD_TO_REVERSE %
%   U:51  REVERSE %
%   B69:1  REVERSED_WORD %
% Rung: 13 %
SOR EQU C5:19.ACC 1 XIO B3:0/3 BST MOV O:2.0 B69:0 NXB JSR U:51 NXB MOV B69:1 N64:91 NXB SWP #N64:91 1 BND EOR
%   C5:19  MODBUS_COIL_CTR %
%   B3:0/3  MODBUS_TEST %
%   B69:0  WORD_TO_REVERSE %
%   U:51  REVERSE %
%   B69:1  REVERSED_WORD %
% Rung: 14 %
SOR EQU C5:19.ACC 2 XIO B3:0/3 BST MOV O:3.0 B69:0 NXB JSR U:51 NXB MOV B69:1 N64:92 NXB SWP #N64:92 1 BND EOR
%   C5:19  MODBUS_COIL_CTR %
%   B3:0/3  MODBUS_TEST %
%   B69:0  WORD_TO_REVERSE %
%   U:51  REVERSE %
%   B69:1  REVERSED_WORD %

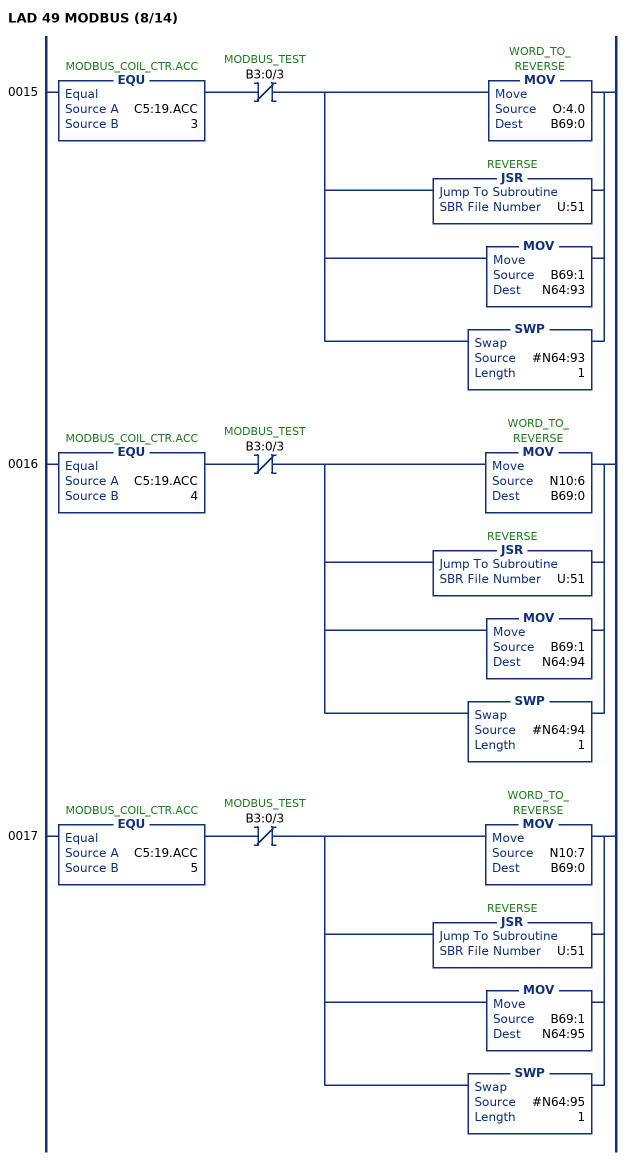
% Rung: 15 %
SOR EQU C5:19.ACC 3 XIO B3:0/3 BST MOV O:4.0 B69:0 NXB JSR U:51 NXB MOV B69:1 N64:93 NXB SWP #N64:93 1 BND EOR
%   C5:19  MODBUS_COIL_CTR %
%   B3:0/3  MODBUS_TEST %
%   B69:0  WORD_TO_REVERSE %
%   U:51  REVERSE %
%   B69:1  REVERSED_WORD %
% Rung: 16 %
SOR EQU C5:19.ACC 4 XIO B3:0/3 BST MOV N10:6 B69:0 NXB JSR U:51 NXB MOV B69:1 N64:94 NXB SWP #N64:94 1 BND EOR
%   C5:19  MODBUS_COIL_CTR %
%   B3:0/3  MODBUS_TEST %
%   N10:6  SYSTEM_ALARMS_0  "ALARM System alarms" %
%   B69:0  WORD_TO_REVERSE %
%   U:51  REVERSE %
%   B69:1  REVERSED_WORD %
% Rung: 17 %
SOR EQU C5:19.ACC 5 XIO B3:0/3 BST MOV N10:7 B69:0 NXB JSR U:51 NXB MOV B69:1 N64:95 NXB SWP #N64:95 1 BND EOR
%   C5:19  MODBUS_COIL_CTR %
%   B3:0/3  MODBUS_TEST %
%   N10:7  SYSTEM_ALARMS_1  "ALARM System alarms" %
%   B69:0  WORD_TO_REVERSE %
%   U:51  REVERSE %
%   B69:1  REVERSED_WORD %

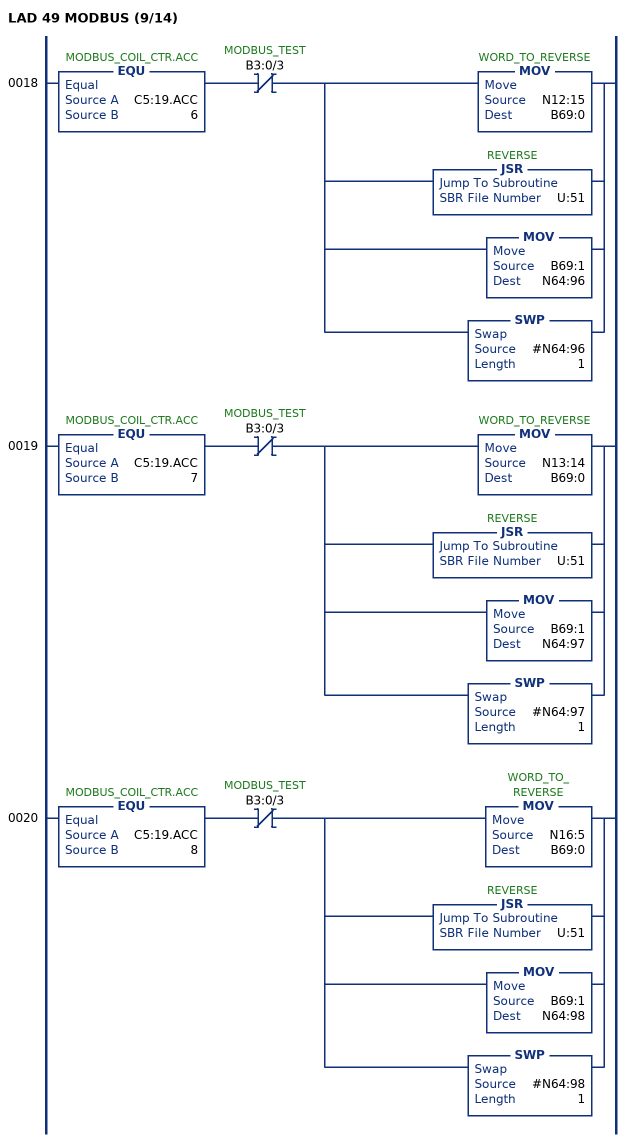
% Rung: 18 %
SOR EQU C5:19.ACC 6 XIO B3:0/3 BST MOV N12:15 B69:0 NXB JSR U:51 NXB MOV B69:1 N64:96 NXB SWP #N64:96 1 BND EOR
%   C5:19  MODBUS_COIL_CTR %
%   B3:0/3  MODBUS_TEST %
%   N12:15  PURIFY_ALARMS_0 %
%   B69:0  WORD_TO_REVERSE %
%   U:51  REVERSE %
%   B69:1  REVERSED_WORD %
% Rung: 19 %
SOR EQU C5:19.ACC 7 XIO B3:0/3 BST MOV N13:14 B69:0 NXB JSR U:51 NXB MOV B69:1 N64:97 NXB SWP #N64:97 1 BND EOR
%   C5:19  MODBUS_COIL_CTR %
%   B3:0/3  MODBUS_TEST %
%   N13:14  REGEN_ALARMS_0 %
%   B69:0  WORD_TO_REVERSE %
%   U:51  REVERSE %
%   B69:1  REVERSED_WORD %
% Rung: 20 %
SOR EQU C5:19.ACC 8 XIO B3:0/3 BST MOV N16:5 B69:0 NXB JSR U:51 NXB MOV B69:1 N64:98 NXB SWP #N64:98 1 BND EOR
%   C5:19  MODBUS_COIL_CTR %
%   B3:0/3  MODBUS_TEST %
%   N16:5  ADS_A_ALARMS_0  "ALARM ADS A Alarms" %
%   B69:0  WORD_TO_REVERSE %
%   U:51  REVERSE %
%   B69:1  REVERSED_WORD %

